ACTION Counter_Reset___entry:
NokCounter:=0;
(*Percent Register löschen*)
i:=0;
FOR i:=1 TO 100 BY 1 DO
  NokPercent[i]:= FALSE;
END_FOR
END_ACTION

ACTION Drehen_links_0_Grad__entry:
MP.ST02.TableData:=PushData(MP.ST02.TableData);
END_ACTION

ACTION Drehen_links_0_Grad__action:
ST02_62_Y6.MoveInit:=TRUE;
END_ACTION

ACTION Drehen_links_0_Grad__exit:
turn_done:=TRUE;
END_ACTION

ACTION Drehen_rechts_180_Grad___entry:
MP.ST02.TableData:=PushData(MP.ST02.TableData);
END_ACTION

ACTION Drehen_rechts_180_Grad___action:
ST02_62_Y6.MoveWork:=TRUE;
END_ACTION

ACTION Drehen_rechts_180_Grad___exit:
turn_done:=TRUE;
END_ACTION

ACTION Msg_Cam_Percent_entry:
MessageHandler.ClearMessageLines(sVisu:=Visu.Message);
END_ACTION

ACTION Msg_Cam_Percent_action:
MessageHandler.Msg.ID:='PM113';
MessageHandler.Msg.Name:='Sensopart Kam.-Erg. Prüfung  n.i.o:';
MessageHandler.Msg.Text:='Sensopart Kam.-Erg. Prüfung  n.i.o:% Fehler';
MessageHandler.Msg.Color:=Color.red;
MessageHandler.Msg.Station:=3;
MessageHandler.MsgButton1Text:='continue';

MessageHandler(
	Prio:=2, 								(*1=highest, .. , 4=lowest*)
	Btn1Addr:=ADR(MsgOk),				(*Address of Button1 , if Zero then Button is unvisible*)
	Btn2Addr:=0(*ADR(MsgCancel)*),			(*Address of Button2 , if Zero then Button is unvisible*)
	sVisu:=Visu.Message);
END_ACTION

ACTION Msg_Cam_Percent_exit:
MsgOk:=FALSE;
MsgCancel:=FALSE;
END_ACTION

ACTION JumpAutoStop__action:
IF ST02_AutoStop.State=STATE_WAIT
THEN
	ST02_AutoStop(Start:=TRUE);
END_IF
END_ACTION

ACTION JumpAutoStop__exit:
ST02_AutoStop.Start:=FALSE;
END_ACTION

ACTION SeqEnd_action:
SFCTime:=TIME_TO_DINT(TIME()-SFCTimeStart);
State:=STATE_WAIT;
END_ACTION

TRANSITION OK:
ST02_35_S31.BitInToCheck
END_TRANSITION

TRANSITION OK_:
NOT MP.ST02.DummyPruefung_93pol
END_TRANSITION

TRANSITION Kamera_betriebsbereit:
(NOT ST02_DT_95_A1.b_kamera_aktiv (*Kamera Farberkennung*)
OR
NOT ST02_DT_95_A1.sm_kamera_nicht_bb) 	 (*Kamera Farberkennung*)
AND
(NOT ST02_DT_95_A2.sm_kamera_nicht_bb
OR
NOT ST02_DT_95_A2.Activated)
END_TRANSITION

TRANSITION Drucker_bereit:
MP.ST02.DummyPruefung_93pol OR
ST00_72_X1_8.BitInToCheck 	(* Tampondrucker Bedruckung ausgeführt oder betriebsbereit *)
END_TRANSITION

TRANSITION MsgOk:
MsgOk OR

ST00_72_X1_8.BitInToCheck 	(* Tampondrucker Bedruckung ausgeführt oder betriebsbereit *)
END_TRANSITION

TRANSITION 180_Grad:
NOT ST02_DT_62_B81.ValveSensor AND	(* Tisch  0 Grad*)
ST02_DT_62_B91.ValveSensor				(* Tisch  180 Grad*)
END_TRANSITION

TRANSITION StateOk:
ST02_62_Y6.State=STATE_OK
AND
gTipImp
END_TRANSITION

TRANSITION nicht leer:
MP.ST02.TableData[2].ProcessData.Part AND

NOT ST02_DT_65B11.BitInToCheck					 (* Tampondrucker Nest 1 leer *)
END_TRANSITION

TRANSITION StateOk:
NOT ST02_Schwenkarm[1].b_180_grad AND
ST02_Schwenkarm[1].b_done
AND
gTipImp
END_TRANSITION

TRANSITION StateOk:
ST02_62_Y17.State=STATE_OK
AND
gTipImp
END_TRANSITION

TRANSITION Drucker_bereit:
NOT MP.ST02.DummyPruefung_93pol AND
ST00_72_X1_8.BitInToCheck 	(* Tampondrucker Bedruckung ausgeführt *)
END_TRANSITION

TRANSITION Drucker_busy:
NOT ST00_72_X1_8.BitInToCheck (* Tampondrucker Bedruckung ausgeführt *)
END_TRANSITION

TRANSITION not_busy:
ST00_72_X1_8.BitInToCheck (* Tampondrucker Bedruckung ausgeführt *)
END_TRANSITION

TRANSITION AutoStop:
		ModeSelect.Mode=MODE_AUTO_STOP
OR	ModeSelect.Mode=MODE_STEP_STOP
END_TRANSITION

TRANSITION Drucker_fertig:
ST00_72_X1_8.BitInToCheck (* Tampondrucker Bedruckung ausgeführt *)
END_TRANSITION

TRANSITION Dummypruefung:
MP.ST02.DummyPruefung_93pol
END_TRANSITION

TRANSITION aktiv:
ST02_DT_95_A1.b_kamera_aktiv (*Kamera Farberkennung*)
OR
ST02_DT_95_A2.Activated	(*Kamera Farberkennung Ethernet*)
END_TRANSITION

TRANSITION Busy:
ST02_DT_95_A1.b_busy	 (*Kamera Farberkennung*)
OR
ST02_DT_95_A2.st_ctrl_out.b_busy (*Kamera Farberkennung Ehternet*)
END_TRANSITION

TRANSITION Done:
(ST02_DT_95_A1.b_done AND	 (*Kamera Farberkennung*)
ST02_DT_95_A1.b_kamera_aktiv AND
((ST02_DT_95_A1.Ergebnis_IO AND NOT ST02_DT_95_A1.Ergebnis_NIO)OR
RepeatCounter>=2 ))
OR
(ST02_DT_95_A2.st_ctrl_out.b_fertig AND
ST02_DT_95_A2.Activated AND
((ST02_DT_95_A2.b_Kam_Pruef_IO AND NOT ST02_DT_95_A2.b_Kam_Pruef_NIO) OR
RepeatCounter>=2))
END_TRANSITION

TRANSITION CamNotAktiv:
(ST02_DT_95_A1.b_done	 (*Kamera Farberkennung*)
AND
NOT ST02_DT_95_A1.b_kamera_aktiv )
OR
(ST02_DT_95_A2.st_ctrl_out.b_fertig  (*Kamera Farberkennung Ethernet*)
AND
NOT ST02_DT_95_A2.Activated)
OR
(NOT ST02_DT_95_A1.b_kamera_aktiv AND NOT ST02_DT_95_A2.Activated)
END_TRANSITION

TRANSITION CamDone:
ST02_DT_95_A1.b_done	 (*Kamera Farberkennung*)
OR
ST02_DT_95_A2.st_ctrl_out.b_fertig	 (*Kamera Farberkennung Ethernet*)
END_TRANSITION

TRANSITION StateOk:
ST02_62_Y17.State=STATE_OK
AND
gTipImp
END_TRANSITION

TRANSITION StateOk:
NOT ST02_Schwenkarm[1].b_0_grad AND
ST02_Schwenkarm[1].b_done
AND
gTipImp
END_TRANSITION

TRANSITION Drucker_bereit:
NOT MP.ST02.DummyPruefung_93pol AND
ST00_72_X1_8.BitInToCheck (* Tampondrucker Bedruckung ausgeführt *)
END_TRANSITION

TRANSITION Drucker_busy:
NOT ST00_72_X1_8.BitInToCheck (* Tampondrucker Bedruckung ausgeführt *)
END_TRANSITION

TRANSITION not_busy:
ST00_72_X1_8.BitInToCheck (* Tampondrucker Bedruckung ausgeführt *)
END_TRANSITION

TRANSITION AutoStop:
		ModeSelect.Mode=MODE_AUTO_STOP
OR	ModeSelect.Mode=MODE_STEP_STOP
END_TRANSITION

TRANSITION Drucker_fertig:
ST00_72_X1_8.BitInToCheck (* Tampondrucker Bedruckung ausgeführt *)
END_TRANSITION

TRANSITION Dummypruefung:
MP.ST02.DummyPruefung_93pol
END_TRANSITION

TRANSITION aktiv:
ST02_DT_95_A1.b_kamera_aktiv (*Kamera Farberkennung*)
OR
ST02_DT_95_A2.Activated(*Kamera Farberkennung Ethernet*)
END_TRANSITION

TRANSITION Busy:
ST02_DT_95_A1.b_busy	 (*Kamera Farberkennung*)
OR
ST02_DT_95_A2.st_ctrl_out.b_busy	(*Kamera Farberkennung Ethernet*)
END_TRANSITION

TRANSITION Done:
ST02_DT_95_A1.b_done AND	 (*Kamera Farberkennung*)
ST02_DT_95_A1.b_kamera_aktiv AND
((ST02_DT_95_A1.Ergebnis_IO AND NOT ST02_DT_95_A1.Ergebnis_NIO)OR
RepeatCounter>=2 )
OR
(ST02_DT_95_A2.st_ctrl_out.b_fertig AND
ST02_DT_95_A2.Activated AND
((ST02_DT_95_A2.b_Kam_Pruef_IO AND NOT ST02_DT_95_A2.b_Kam_Pruef_NIO) OR
RepeatCounter>=2))
END_TRANSITION

TRANSITION CamNotAktiv:
(ST02_DT_95_A1.b_done	 (*Kamera Farberkennung*)
AND
NOT ST02_DT_95_A1.b_kamera_aktiv)
OR
(ST02_DT_95_A2.st_ctrl_out.b_fertig  (*Kamera Farberkennung Ethernet*)
AND
NOT ST02_DT_95_A2.Activated)
END_TRANSITION

TRANSITION CamDone:
ST02_DT_95_A1.b_done	 (*Kamera Farberkennung*)
OR
ST02_DT_95_A2.st_ctrl_out.b_fertig	 (*Kamera Farberkennung Ethernet*)
END_TRANSITION

TRANSITION StateOk:
NOT ST02_Schwenkarm[1].b_90_grad AND
ST02_Schwenkarm[1].b_done
AND
gTipImp
END_TRANSITION

TRANSITION 0_Grad:
ST02_DT_62_B81.ValveSensor AND	(* Tisch 0 Grad*)
NOT ST02_DT_62_B91.ValveSensor	(* Tisch 180 Grad*)
END_TRANSITION

TRANSITION StateOk:
ST02_62_Y6.State=STATE_OK
AND
gTipImp
END_TRANSITION

TRANSITION nicht leer:
MP.ST02.TableData[2].ProcessData.Part AND

NOT ST02_DT_65B21.BitInToCheck					 (* Tampondrucker Nest 2 leer *)
END_TRANSITION

TRANSITION StateOk:
NOT ST02_Schwenkarm[2].b_180_grad AND
ST02_Schwenkarm[2].b_done
AND
gTipImp
END_TRANSITION

TRANSITION StateOk:
ST02_62_Y18.State=STATE_OK
AND
gTipImp
END_TRANSITION

TRANSITION Drucker_bereit:
NOT MP.ST02.DummyPruefung_93pol AND
ST00_72_X1_8.BitInToCheck (* Tampondrucker Bedruckung ausgeführt *)
END_TRANSITION

TRANSITION Drucker_busy:
NOT ST00_72_X1_8.BitInToCheck (* Tampondrucker Bedruckung ausgeführt *)
END_TRANSITION

TRANSITION not_busy:
ST00_72_X1_8.BitInToCheck (* Tampondrucker Bedruckung ausgeführt *)
END_TRANSITION

TRANSITION AutoStop:
		ModeSelect.Mode=MODE_AUTO_STOP
OR	ModeSelect.Mode=MODE_STEP_STOP
END_TRANSITION

TRANSITION Drucker_fertig:
ST00_72_X1_8.BitInToCheck (* Tampondrucker Bedruckung ausgeführt *)
END_TRANSITION

TRANSITION Dummypruefung:
MP.ST02.DummyPruefung_93pol
END_TRANSITION

TRANSITION aktiv:
ST02_DT_95_A1.b_kamera_aktiv (*Kamera Farberkennung*)
OR
ST02_DT_95_A2.Activated	(*Kamera Farberkennung Ethernet*)
END_TRANSITION

TRANSITION Busy:
ST02_DT_95_A1.b_busy	 (*Kamera Farberkennung*)
OR
ST02_DT_95_A2.st_ctrl_out.b_busy (*Kamera Farberkennung Ehternet*)
END_TRANSITION

TRANSITION Done:
(ST02_DT_95_A1.b_done AND	 (*Kamera Farberkennung*)
ST02_DT_95_A1.b_kamera_aktiv AND
((ST02_DT_95_A1.Ergebnis_IO AND NOT ST02_DT_95_A1.Ergebnis_NIO)OR
RepeatCounter>=2))
OR
(ST02_DT_95_A2.st_ctrl_out.b_fertig AND
ST02_DT_95_A2.Activated AND
((ST02_DT_95_A2.b_Kam_Pruef_IO AND NOT ST02_DT_95_A2.b_Kam_Pruef_NIO) OR
RepeatCounter>=2))
END_TRANSITION

TRANSITION CamNotAktiv:
(ST02_DT_95_A1.b_done	 (*Kamera Farberkennung*)
AND
NOT ST02_DT_95_A1.b_kamera_aktiv)
OR
(ST02_DT_95_A2.st_ctrl_out.b_fertig  (*Kamera Farberkennung Ethernet*)
AND
NOT ST02_DT_95_A2.Activated)
END_TRANSITION

TRANSITION CamDone:
ST02_DT_95_A1.b_done	 (*Kamera Farberkennung*)
OR
ST02_DT_95_A2.st_ctrl_out.b_fertig	 (*Kamera Farberkennung Ethernet*)
END_TRANSITION

TRANSITION StateOk:
ST02_62_Y18.State=STATE_OK
AND
gTipImp
END_TRANSITION

TRANSITION StateOk:
NOT ST02_Schwenkarm[2].b_0_grad AND
ST02_Schwenkarm[2].b_done
AND
gTipImp
END_TRANSITION

TRANSITION Drucker_bereit:
NOT MP.ST02.DummyPruefung_93pol AND
ST00_72_X1_8.BitInToCheck (* Tampondrucker Bedruckung ausgeführt *)
END_TRANSITION

TRANSITION Drucker_busy:
NOT ST00_72_X1_8.BitInToCheck (* Tampondrucker Bedruckung ausgeführt *)
END_TRANSITION

TRANSITION not_busy:
ST00_72_X1_8.BitInToCheck (* Tampondrucker Bedruckung ausgeführt *)
END_TRANSITION

TRANSITION AutoStop:
		ModeSelect.Mode=MODE_AUTO_STOP
OR	ModeSelect.Mode=MODE_STEP_STOP
END_TRANSITION

TRANSITION Drucker_fertig:
ST00_72_X1_8.BitInToCheck (* Tampondrucker Bedruckung ausgeführt *)
END_TRANSITION

TRANSITION Dummypruefung:
MP.ST02.DummyPruefung_93pol
END_TRANSITION

TRANSITION aktiv:
ST02_DT_95_A1.b_kamera_aktiv (*Kamera Farberkennung*)
OR
ST02_DT_95_A2.Activated (*Kamera Farberkennung Ethernet*)
END_TRANSITION

TRANSITION Busy:
ST02_DT_95_A1.b_busy	 (*Kamera Farberkennung*)
OR
ST02_DT_95_A2.st_ctrl_out.b_busy	(*Kamera Farberkennung Ethernet*)
END_TRANSITION

TRANSITION Done:
(ST02_DT_95_A1.b_done AND	 (*Kamera Farberkennung*)
ST02_DT_95_A1.b_kamera_aktiv AND
((ST02_DT_95_A1.Ergebnis_IO AND NOT ST02_DT_95_A1.Ergebnis_NIO)OR
RepeatCounter>=2 ))
OR
(ST02_DT_95_A2.st_ctrl_out.b_fertig AND
ST02_DT_95_A2.Activated AND
((ST02_DT_95_A2.b_Kam_Pruef_IO AND NOT ST02_DT_95_A2.b_Kam_Pruef_NIO) OR
RepeatCounter>=2))
END_TRANSITION

TRANSITION CamNotAktiv:
(ST02_DT_95_A1.b_done	 (*Kamera Farberkennung*)
AND
NOT ST02_DT_95_A1.b_kamera_aktiv)
OR
(ST02_DT_95_A2.st_ctrl_out.b_fertig  (*Kamera Farberkennung Ethernet*)
AND
NOT ST02_DT_95_A2.Activated)
END_TRANSITION

TRANSITION CamDone:
ST02_DT_95_A1.b_done	 (*Kamera Farberkennung*)
OR
ST02_DT_95_A2.st_ctrl_out.b_fertig	 (*Kamera Farberkennung Ethernet*)
END_TRANSITION

TRANSITION StateOk:
NOT ST02_Schwenkarm[2].b_90_grad AND
ST02_Schwenkarm[2].b_done
AND
 (gTipImp OR ModeSelect.Mode=MODE_MANUAL)
END_TRANSITION

TRANSITION CounterOK:
NOT MP.ST02.DummyPruefung_93pol AND
NokCounter<MP.ST02.CamNoOfErrors AND
NokCounterPercent < MP.ST02.CamNoOfErrorsPercent
OR
( MP.ST02.DummyPruefung_93pol AND
LoopCounter < 6)
END_TRANSITION

TRANSITION Nok_Cont:
NOT MP.ST02.DummyPruefung_93pol AND
NokCounter >= MP.ST02.CamNoOfErrors
END_TRANSITION

TRANSITION Nok_Percent:
NOT MP.ST02.DummyPruefung_93pol AND
NokCounterPercent >= MP.ST02.CamNoOfErrorsPercent
END_TRANSITION

TRANSITION Dummytest:
 MP.ST02.DummyPruefung_93pol AND
LoopCounter = 6
END_TRANSITION

TRANSITION Robo_free:
Robot01.ActualArea <> 3
END_TRANSITION

TRANSITION 180_Grad_:
NOT ST02_DT_62_B81.ValveSensor AND	(* Tisch  0 Grad*)
ST02_DT_62_B91.ValveSensor				(* Tisch  180 Grad*)
END_TRANSITION

TRANSITION StateOk:
ST02_62_Y6.State=STATE_OK
AND
gTipImp
END_TRANSITION

TRANSITION 0_Grad_:
ST02_DT_62_B81.ValveSensor AND	(* Tisch 0 Grad*)
NOT ST02_DT_62_B91.ValveSensor	(* Tisch 180 Grad*)
END_TRANSITION

TRANSITION StateOk:
ST02_62_Y6.State=STATE_OK
AND
gTipImp
END_TRANSITION

TRANSITION end:
NOT MP.ST02.DummyPruefung_93pol
END_TRANSITION

TRANSITION AutoRun:
(ModeSelect.Mode=MODE_AUTO_RUN OR
ModeSelect.Mode=MODE_STEP_RUN)
OR (SpecialMode06.State=State_Run AND
		(gTypeCode=312 OR			(*93pol*)
		gTypeCode=499))				(*102pol*)
END_TRANSITION

TRANSITION AutoStop:
ModeSelect.Mode=MODE_AUTO_STOP OR
ModeSelect.Mode=MODE_STEP_STOP
END_TRANSITION

TRANSITION StateOk:
ST02_AutoStop.State=STATE_OK
END_TRANSITION
END_PROGRAM

(* POU Stations/ST_02_RT_Tampondrucker/ST02_SFCs/ST02_AutoStop, SFC *)
PROGRAM ST02_AutoStop

VAR_OUTPUT
	SFCCurrentPOU			: STRING:='ST02_AutoStop';
	SFCCurrentStep			: STRING:='';
	SFCTime					: DINT;
	State   				: StateObject	:= STATE_WAIT;
	Result  				: StateResult;
END_VAR
VAR_INPUT
	Start					: BOOL;
END_VAR
VAR
	MsgOK					: BOOL;
	MsgCancel				: BOOL;
	SFCRun					: BOOL;
	SFCTimeStart			: TIME;
	(* Userdefinded area *)

END_VAR
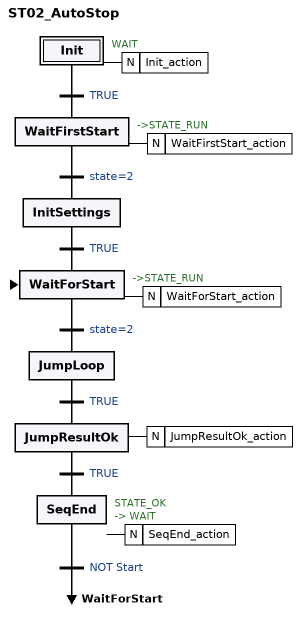
INITIAL_STEP Init: (* WAIT *)
	Init_action(N);
END_STEP
TRANSITION FROM Init TO WaitFirstStart := TRUE;
END_TRANSITION
STEP WaitFirstStart: (* ->STATE_RUN *)
	WaitFirstStart_action(N);
END_STEP
TRANSITION FROM WaitFirstStart TO InitSettings := state=2;
END_TRANSITION
STEP InitSettings:
END_STEP
TRANSITION FROM InitSettings TO WaitForStart := TRUE;
END_TRANSITION
STEP WaitForStart: (* ->STATE_RUN *)
	WaitForStart_action(N);
END_STEP
TRANSITION FROM WaitForStart TO JumpLoop := state=2;
END_TRANSITION
STEP JumpLoop:
END_STEP
TRANSITION FROM JumpLoop TO JumpResultOk := TRUE;
END_TRANSITION
STEP JumpResultOk:
	JumpResultOk_action(N);
END_STEP
TRANSITION FROM JumpResultOk TO SeqEnd := TRUE;
END_TRANSITION
STEP SeqEnd: (* STATE_OK / -> WAIT *)
	SeqEnd_action(N);
END_STEP
TRANSITION FROM SeqEnd TO WaitForStart := NOT Start;
END_TRANSITION

ACTION Init_action:
Start:=FALSE;
State:=STATE_WAIT;
MsgOK:=FALSE;
MsgCancel:=FALSE;
SFCRun:=FALSE;
END_ACTION

ACTION WaitFirstStart_action:
IF Start
THEN
	State:=STATE_RUN;
	Result:=RESULT_NON;
(*ELSE*)
END_IF
END_ACTION

ACTION WaitForStart_action:
IF Start
THEN
	State:=STATE_RUN;
	Result:=RESULT_NON;
	SFCTimeStart:=TIME();
END_IF
END_ACTION

ACTION JumpResultOk_action:
Result:=RESULT_OK;
END_ACTION

ACTION SeqEnd_action:
IF 	State=STATE_RUN THEN
	SFCTime:=TIME_TO_DINT(TIME()-SFCTimeStart);
	State:=STATE_OK;
END_IF

IF 	NOT Start THEN
	State:=STATE_WAIT;
END_IF
END_ACTION
END_PROGRAM

(* POU Stations/ST_03_Ruestsaetze/ST_03_SFCs/Zufuehrungen/ST03_102pol_Zufuehrung, SFC *)
 PROGRAM ST03_102pol_Zufuehrung
VAR_OUTPUT
	SFCCurrentPOU			: STRING:='ST03_102pol_Zufuehrung';
	SFCCurrentStep			: STRING:='';
	FB_CurrentStepHistorie	: FB_CurrentStepHistorie;
	SFCTime					: DINT;
	State   				: StateObject	:= STATE_WAIT;
END_VAR
VAR_INPUT
	Start				: BOOL;
	Result  			: DINT;
END_VAR
VAR
	MsgOK				: BOOL;
	MsgCancel			: BOOL;
	SFCRun				: BOOL;
	SFCTimeStart		: TIME;
	(* Userdefinded area *)
	i					: INT;
	PartReady			: BOOL;

	ResultBufferIFM		: ARRAY[1..10] OF BOOL;
	LoopCounter			: DINT;	(* Anzahl Dummy *)
	Dummy_test_Result	: BOOL;
	Delay				: TON;
END_VAR
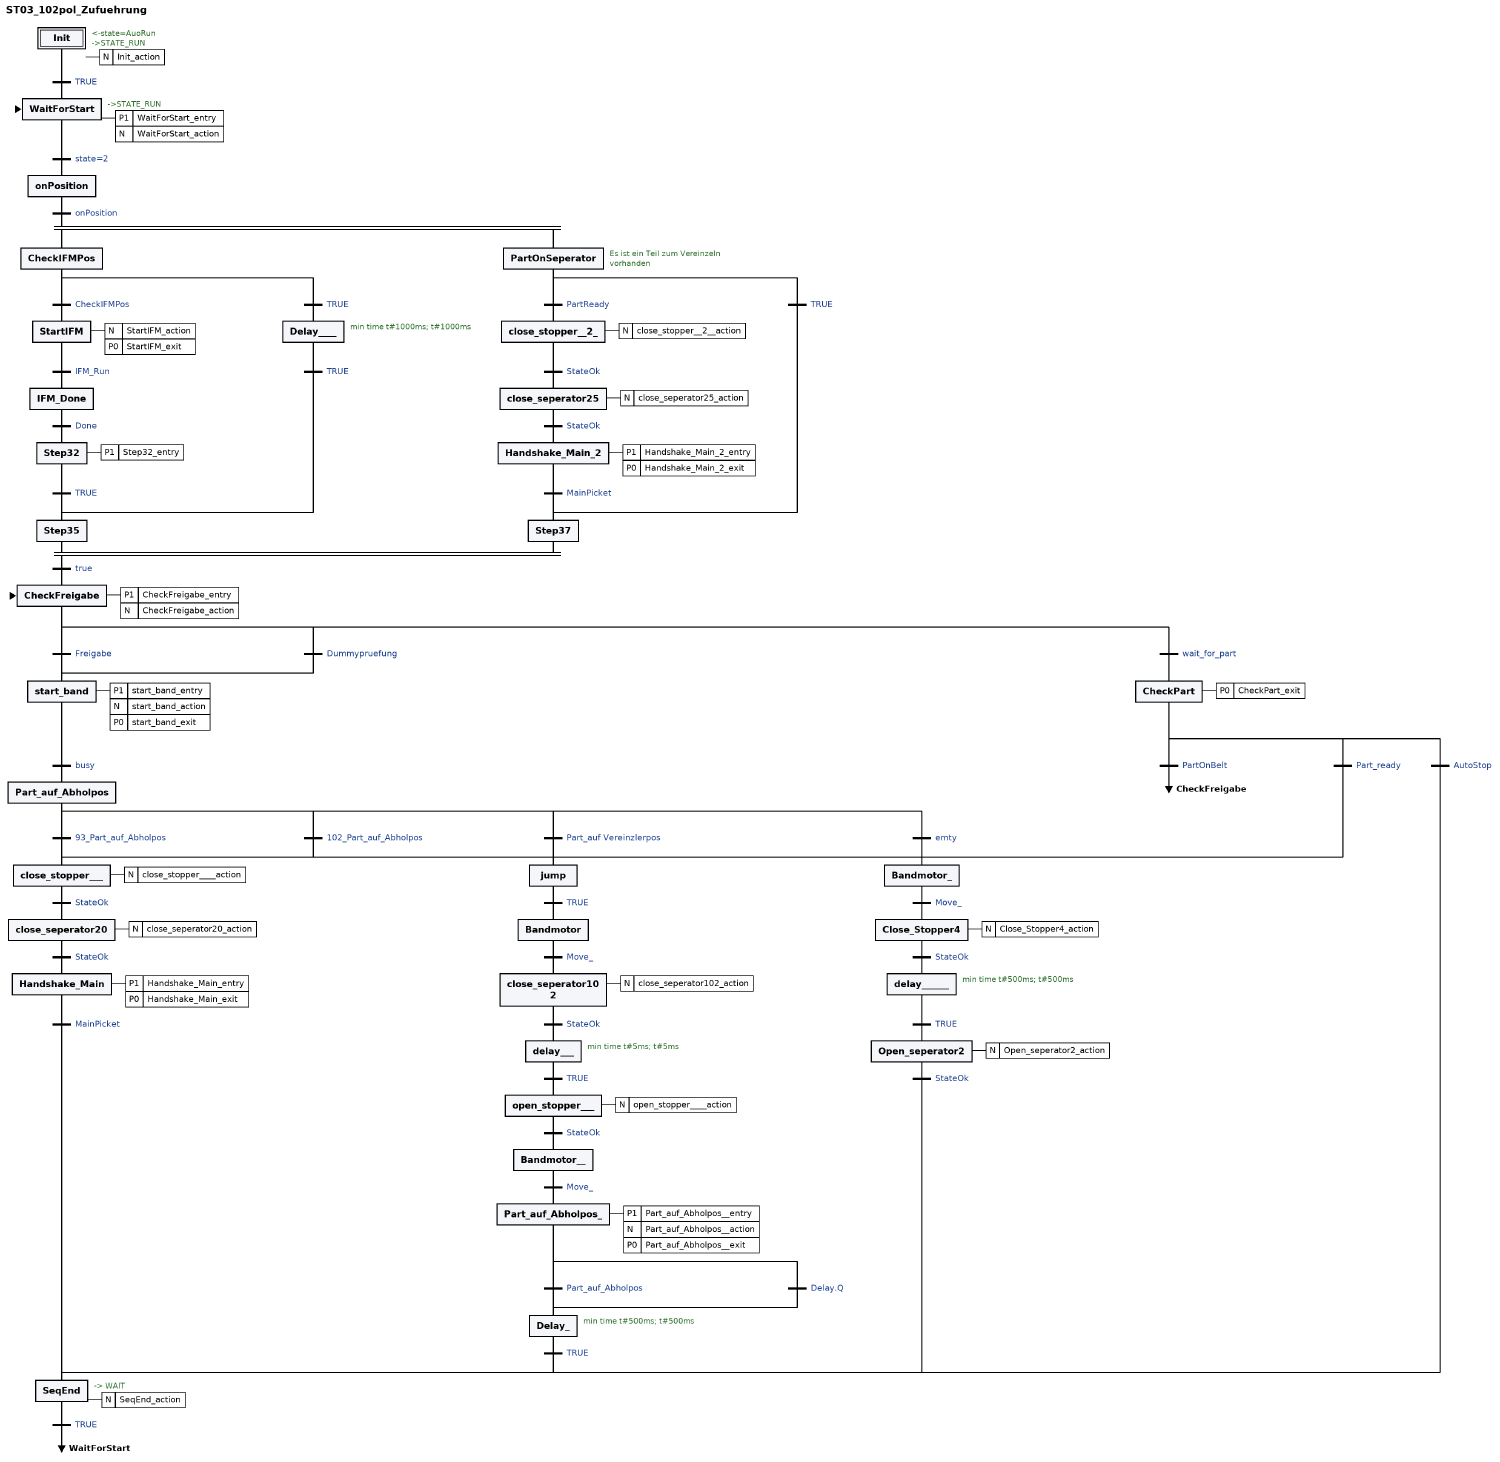
INITIAL_STEP Init: (* <-state=AuoRun / ->STATE_RUN *)
	Init_action(N);
END_STEP
TRANSITION FROM Init TO WaitForStart := TRUE;
END_TRANSITION
STEP WaitForStart: (* ->STATE_RUN *)
	WaitForStart_entry(P1);
	WaitForStart_action(N);
END_STEP
TRANSITION FROM WaitForStart TO onPosition := state=2;
END_TRANSITION
STEP onPosition:
END_STEP
TRANSITION FROM onPosition TO (CheckIFMPos, PartOnSeperator) := onPosition;
END_TRANSITION
STEP CheckIFMPos:
END_STEP
TRANSITION FROM CheckIFMPos TO StartIFM := CheckIFMPos;
END_TRANSITION
TRANSITION FROM CheckIFMPos TO Delay____ := TRUE;
END_TRANSITION
STEP Delay____: (* min time t#1000ms; t#1000ms *)
END_STEP
TRANSITION FROM Delay____ TO Step35 := TRUE;
END_TRANSITION
STEP StartIFM:
	StartIFM_action(N);
	StartIFM_exit(P0);
END_STEP
TRANSITION FROM StartIFM TO IFM_Done := IFM_Run;
END_TRANSITION
STEP IFM_Done:
END_STEP
TRANSITION FROM IFM_Done TO Step32 := Done;
END_TRANSITION
STEP Step32:
	Step32_entry(P1);
END_STEP
TRANSITION FROM Step32 TO Step35 := TRUE;
END_TRANSITION
STEP Step35:
END_STEP
STEP PartOnSeperator: (* Es ist ein Teil zum Vereinzeln vorhanden *)
END_STEP
TRANSITION FROM PartOnSeperator TO close_stopper__2_ := PartReady;
END_TRANSITION
TRANSITION FROM PartOnSeperator TO Step37 := TRUE;
END_TRANSITION
STEP close_stopper__2_:
	close_stopper__2__action(N);
END_STEP
TRANSITION FROM close_stopper__2_ TO close_seperator25 := StateOk;
END_TRANSITION
STEP close_seperator25:
	close_seperator25_action(N);
END_STEP
TRANSITION FROM close_seperator25 TO Handshake_Main_2 := StateOk;
END_TRANSITION
STEP Handshake_Main_2:
	Handshake_Main_2_entry(P1);
	Handshake_Main_2_exit(P0);
END_STEP
TRANSITION FROM Handshake_Main_2 TO Step37 := MainPicket;
END_TRANSITION
STEP Step37:
END_STEP
TRANSITION FROM (Step35, Step37) TO CheckFreigabe := true;
END_TRANSITION
STEP CheckFreigabe:
	CheckFreigabe_entry(P1);
	CheckFreigabe_action(N);
END_STEP
TRANSITION FROM CheckFreigabe TO start_band := Freigabe;
END_TRANSITION
TRANSITION FROM CheckFreigabe TO start_band := Dummypruefung;
END_TRANSITION
TRANSITION FROM CheckFreigabe TO CheckPart := wait_for_part;
END_TRANSITION
STEP CheckPart:
	CheckPart_exit(P0);
END_STEP
TRANSITION FROM CheckPart TO CheckFreigabe := PartOnBelt;
END_TRANSITION
TRANSITION FROM CheckPart TO close_stopper___ := Part_ready;
END_TRANSITION
TRANSITION FROM CheckPart TO SeqEnd := AutoStop;
END_TRANSITION
STEP start_band:
	start_band_entry(P1);
	start_band_action(N);
	start_band_exit(P0);
END_STEP
TRANSITION FROM start_band TO Part_auf_Abholpos := busy;
END_TRANSITION
STEP Part_auf_Abholpos:
END_STEP
TRANSITION FROM Part_auf_Abholpos TO close_stopper___ := 93_Part_auf_Abholpos;
END_TRANSITION
TRANSITION FROM Part_auf_Abholpos TO close_stopper___ := 102_Part_auf_Abholpos;
END_TRANSITION
TRANSITION FROM Part_auf_Abholpos TO jump := Part_auf Vereinzlerpos;
END_TRANSITION
TRANSITION FROM Part_auf_Abholpos TO Bandmotor_ := emty;
END_TRANSITION
STEP jump:
END_STEP
TRANSITION FROM jump TO Bandmotor := TRUE;
END_TRANSITION
STEP Bandmotor:
END_STEP
TRANSITION FROM Bandmotor TO close_seperator102 := Move_;
END_TRANSITION
STEP close_seperator102:
	close_seperator102_action(N);
END_STEP
TRANSITION FROM close_seperator102 TO delay___ := StateOk;
END_TRANSITION
STEP delay___: (* min time t#5ms; t#5ms *)
END_STEP
TRANSITION FROM delay___ TO open_stopper___ := TRUE;
END_TRANSITION
STEP open_stopper___:
	open_stopper____action(N);
END_STEP
TRANSITION FROM open_stopper___ TO Bandmotor__ := StateOk;
END_TRANSITION
STEP Bandmotor__:
END_STEP
TRANSITION FROM Bandmotor__ TO Part_auf_Abholpos_ := Move_;
END_TRANSITION
STEP Part_auf_Abholpos_:
	Part_auf_Abholpos__entry(P1);
	Part_auf_Abholpos__action(N);
	Part_auf_Abholpos__exit(P0);
END_STEP
TRANSITION FROM Part_auf_Abholpos_ TO Delay_ := Part_auf_Abholpos;
END_TRANSITION
TRANSITION FROM Part_auf_Abholpos_ TO Delay_ := Delay.Q;
END_TRANSITION
STEP Delay_: (* min time t#500ms; t#500ms *)
END_STEP
TRANSITION FROM Delay_ TO SeqEnd := TRUE;
END_TRANSITION
STEP Bandmotor_:
END_STEP
TRANSITION FROM Bandmotor_ TO Close_Stopper4 := Move_;
END_TRANSITION
STEP Close_Stopper4:
	Close_Stopper4_action(N);
END_STEP
TRANSITION FROM Close_Stopper4 TO delay______ := StateOk;
END_TRANSITION
STEP delay______: (* min time t#500ms; t#500ms *)
END_STEP
TRANSITION FROM delay______ TO Open_seperator2 := TRUE;
END_TRANSITION
STEP Open_seperator2:
	Open_seperator2_action(N);
END_STEP
TRANSITION FROM Open_seperator2 TO SeqEnd := StateOk;
END_TRANSITION
STEP close_stopper___:
	close_stopper____action(N);
END_STEP
TRANSITION FROM close_stopper___ TO close_seperator20 := StateOk;
END_TRANSITION
STEP close_seperator20:
	close_seperator20_action(N);
END_STEP
TRANSITION FROM close_seperator20 TO Handshake_Main := StateOk;
END_TRANSITION
STEP Handshake_Main:
	Handshake_Main_entry(P1);
	Handshake_Main_exit(P0);
END_STEP
TRANSITION FROM Handshake_Main TO SeqEnd := MainPicket;
END_TRANSITION
STEP SeqEnd: (* -> WAIT *)
	SeqEnd_action(N);
END_STEP
TRANSITION FROM SeqEnd TO WaitForStart := TRUE;
END_TRANSITION

ACTION Init_action:
Start:=FALSE;
State:=STATE_WAIT;
MsgOK:=FALSE;
MsgCancel:=FALSE;
SFCRun:=FALSE;
Result:=RESULT_NON;
PartReady := FALSE;
ST03_Band.fb_ton_Stopp_Band.IN:=FALSE;
LoopCounter :=0;
END_ACTION

ACTION WaitForStart_entry:
;
END_ACTION

ACTION WaitForStart_action:
IF 	Start   THEN
	State:=STATE_RUN;
	Result:=RESULT_NON;
	SFCTimeStart:=TIME();
	Start:=FALSE;
ELSE
	State:=STATE_WAIT;
	MsgOK:=FALSE;
	MsgCancel:=FALSE;
	SFCRun:=FALSE;
END_IF
END_ACTION

ACTION StartIFM_action:
ST03_IFM_Camera.Start:=TRUE;
END_ACTION

ACTION StartIFM_exit:
ST03_IFM_Camera.Start:=FALSE;
END_ACTION

ACTION Step32_entry:
IF ST02_FDB_55X1_6_IO.BitInToCheck AND
ST02_FDB_56X1_6_IO.BitInToCheck
THEN
   Dummy_test_Result:=TRUE;
ELSE
   Dummy_test_Result:=FALSE;
END_IF

(*Ergebnise in Puffer eintragen für Dummyprüfung IFM Kamera*)
i:=0;
FOR i:=10 TO 2 BY-1 DO
	ResultBufferIFM[i]:=ResultBufferIFM[i-1];
END_FOR
ResultBufferIFM[1]:=Dummy_test_Result;
END_ACTION

ACTION close_stopper__2__action:
ST00_74_Y2_4.MoveInit:=TRUE;
END_ACTION

ACTION close_seperator25_action:
ST00_74_Y2_5.MoveWork:=TRUE;
END_ACTION

ACTION Handshake_Main_2_entry:
PartReady := TRUE;
END_ACTION

ACTION Handshake_Main_2_exit:
PartReady := FALSE;
END_ACTION

ACTION CheckFreigabe_entry:
LoopCounter := LoopCounter +1;
END_ACTION

ACTION CheckFreigabe_action:
IF MP.ST02.DummyPruefung_93pol THEN
ST03_BG3_X53_0.SetSignalHigh := TRUE; (*LED Taster Start Band Dummyprüfung*)
END_IF
END_ACTION

ACTION CheckPart_exit:
ST03_Band.fb_ton_Stopp_Band.IN:=FALSE;
END_ACTION

ACTION start_band_entry:
IF NOT MP.ST02.DummyPruefung_93pol THEN
			ST03_51_M1.sVelo.maxRpm;
			ST03_51_M1.Vorgabe_Velo:=32000; 			(*mm/min*)
			ST03_51_M1.Vorgabe_Pos_Rel:=MP.ST02.IFMPos;
			ST03_51_M1.MoveRel:=TRUE;
ELSE
			ST03_51_M1.sVelo.maxRpm;
			ST03_51_M1.Vorgabe_Velo:=16000; 			(*mm/min*)
			ST03_51_M1.Vorgabe_Pos_Rel:=MP.ST02.IFMPosDummy;
			ST03_51_M1.MoveRel:=TRUE;
END_IF


ST03_Band.fb_ton_Stopp_Band.IN:=TRUE;
END_ACTION

ACTION start_band_action:
ST03_BG3_X53_0.SetSignalLow := TRUE; (*LED Taster Start Band Dummyprüfung*)
END_ACTION

ACTION start_band_exit:
ST03_51_M1.MoveRel:=FALSE;
END_ACTION

ACTION close_seperator102_action:
ST00_74_Y2_5.MoveWork:=TRUE;
END_ACTION

ACTION open_stopper____action:
ST00_74_Y2_4.MoveWork:=TRUE;
END_ACTION

ACTION Part_auf_Abholpos__entry:
Delay(IN:=FALSE);
END_ACTION

ACTION Part_auf_Abholpos__action:
Delay(IN:=TRUE, PT:=t#2s);
END_ACTION

ACTION Part_auf_Abholpos__exit:
Delay(IN:=FALSE);
END_ACTION

ACTION Close_Stopper4_action:
ST00_74_Y2_4.MoveInit:=TRUE;
END_ACTION

ACTION Open_seperator2_action:
ST00_74_Y2_5.MoveInit:=TRUE;
END_ACTION

ACTION close_stopper____action:
ST00_74_Y2_4.MoveInit:=TRUE;
END_ACTION

ACTION close_seperator20_action:
ST00_74_Y2_5.MoveWork:=TRUE;
END_ACTION

ACTION Handshake_Main_entry:
PartReady := TRUE;
END_ACTION

ACTION Handshake_Main_exit:
PartReady := FALSE;
END_ACTION

ACTION SeqEnd_action:
SFCTime:=TIME_TO_DINT(TIME()-SFCTimeStart);
State:=STATE_WAIT;
END_ACTION

TRANSITION onPosition:
ST03_51_M1.On_Position
END_TRANSITION

TRANSITION CheckIFMPos:
(MP.ST00.IFMCameraActive AND NOT MP.ST02.DummyPruefung_93pol)
OR
(MP.ST02.DummyPruefung_93pol AND
LoopCounter <= 6)
END_TRANSITION

TRANSITION IFM_Run:
ST03_IFM_Camera.State = STATE_RUN
END_TRANSITION

TRANSITION Done:
ST03_IFM_Camera.State = STATE_WAIT
END_TRANSITION

TRANSITION PartReady:
(gTypeCode=4991 AND				(*102pol*)
 ST02_FDB_80_B02.BitInToCheck)	(*Entnahmeposition 2*)
OR
(gTypeCode=312 AND				(*93pol*)
 ST00_72_X1_3.BitInToCheck) 	(*Schnittstelle Tampondrucker Teil in Abholposition; Band Entnahmeposition 1*)
END_TRANSITION

TRANSITION StateOk:
ST00_74_Y2_4.State=STATE_OK
END_TRANSITION

TRANSITION StateOk:
ST00_74_Y2_5.State=STATE_OK
END_TRANSITION

TRANSITION MainPicket:
ST03_Main.Nest_Empty
END_TRANSITION

TRANSITION Freigabe:
NOT MP.ST02.DummyPruefung_93pol AND
NOT ST02_S1_40K01.BitInToCheck AND			(* Freigabe Förderband von SPM*)
NOT ST00_73_K4.BitInToCheck AND
(*Robot01.ActualArea <> 4	AND*)								(*  ISK anwesend am Vereinzler*)
NOT ST03_Band.fb_ton_Stopp_Band.Q
END_TRANSITION

TRANSITION Dummypruefung:
(SpecialMode06.StartErlaubt93pol AND
MP.ST02.DummyPruefung_93pol AND
NOT ST03_Band.fb_ton_Stopp_Band.Q AND
ST03_BG3_S53_0.BitInToCheck) (*Taster Start Band Dummyprüfung*)
OR
(SpecialMode06.StartErlaubt93pol AND
MP.ST02.DummyPruefung_93pol AND
LoopCounter >= 7 AND
NOT ST03_Band.fb_ton_Stopp_Band.Q)
END_TRANSITION

TRANSITION wait_for_part:
NOT MP.ST02.DummyPruefung_93pol
END_TRANSITION

TRANSITION PartOnBelt:
NOT ST02_FDB_40_B61.BitInToCheck
END_TRANSITION

TRANSITION Part_ready:
(gTypeCode=312 AND				(*93pol*)
 ST00_72_X1_3.BitInToCheck) 	(*Schnittstelle Tampondrucker Teil in Abholposition, Band Entnahmeposition 1 *)
OR
(gTypeCode=4991 AND				(*102pol*)
 ST02_FDB_80_B02.BitInToCheck)	(*Entnahmeposition 2*)
END_TRANSITION

TRANSITION AutoStop:
ModeSelect.Mode=MODE_AUTO_STOP OR
ModeSelect.Mode=MODE_STEP_STOP
END_TRANSITION

TRANSITION busy:
ST03_51_M1.Busy
END_TRANSITION

TRANSITION 93_Part_auf_Abholpos:
gTypeCode=312 AND			(*93pol*)
ST00_72_X1_3.BitInToCheck	(*Schnittstelle Tampondrucker Teil in Abholposition, Band Entnahmeposition 1 *)
END_TRANSITION

TRANSITION 102_Part_auf_Abholpos:
gTypeCode=4991 AND				(*102pol*)
ST02_FDB_80_B02.BitInToCheck	(*Entnahmeposition 2*)
END_TRANSITION

TRANSITION Part_auf Vereinzlerpos:
ST00_72_X1_3.BitInToCheck (* Schnittstelle Tampondrucker Teil in Abholposition *) (* Band Entnahmeposition 1 *)
END_TRANSITION

TRANSITION Move_:
NOT ST03_51_M1.On_Position
END_TRANSITION

TRANSITION StateOk:
ST00_74_Y2_5.State=STATE_OK
END_TRANSITION

TRANSITION StateOk:
ST00_74_Y2_4.State=STATE_OK
END_TRANSITION

TRANSITION Move_:
NOT ST03_51_M1.On_Position
END_TRANSITION

TRANSITION Part_auf_Abholpos:
ST02_FDB_80_B02.BitInToCheck 		(*Entnahmeposition 2*)
END_TRANSITION

TRANSITION emty:
NOT ST00_72_X1_3.BitInToCheck (* Schnittstelle Tampondrucker Teil in Abholposition *) (* Band Entnahmeposition 1 *)
END_TRANSITION

TRANSITION Move_:
NOT ST03_51_M1.On_Position
END_TRANSITION

TRANSITION StateOk:
ST00_74_Y2_4.State=STATE_OK
END_TRANSITION

TRANSITION StateOk:
ST00_74_Y2_5.State=STATE_OK
END_TRANSITION

TRANSITION StateOk:
ST00_74_Y2_4.State=STATE_OK
END_TRANSITION

TRANSITION StateOk:
ST00_74_Y2_5.State=STATE_OK
END_TRANSITION

TRANSITION MainPicket:
ST03_Main.Nest_Empty
END_TRANSITION
END_PROGRAM

(* POU Stations/ST_03_Ruestsaetze/ST_03_SFCs/ST03_IFM_Camera, SFC *)
PROGRAM ST03_IFM_Camera
VAR_OUTPUT
	SFCCurrentPOU		: STRING:='ST03_IFM_Camera';
	SFCCurrentStep		: STRING:='';
	FB_CurrentStepHistorie: FB_CurrentStepHistorie;
	SFCTime				: DINT;
	State   			: StateObject	:= STATE_WAIT;
	Result  			: StateResult;
END_VAR
VAR_INPUT
	Start				: BOOL;
END_VAR
VAR
	MsgOK				: BOOL;
	MsgCancel			: BOOL;
	SFCRun				: BOOL;
	SFCTimeStart		: TIME;
	fb_r_trig_start		: R_TRIG;
	Error				: ErrorStruct;
	(* Userdefinded area *)
	PartReady      		: BOOL;
 	ErrorSep        	: BOOL;
	NokCounter    		: DINT;
	WdhCounter   		: DINT;
	oldPosition			: LREAL;
END_VAR
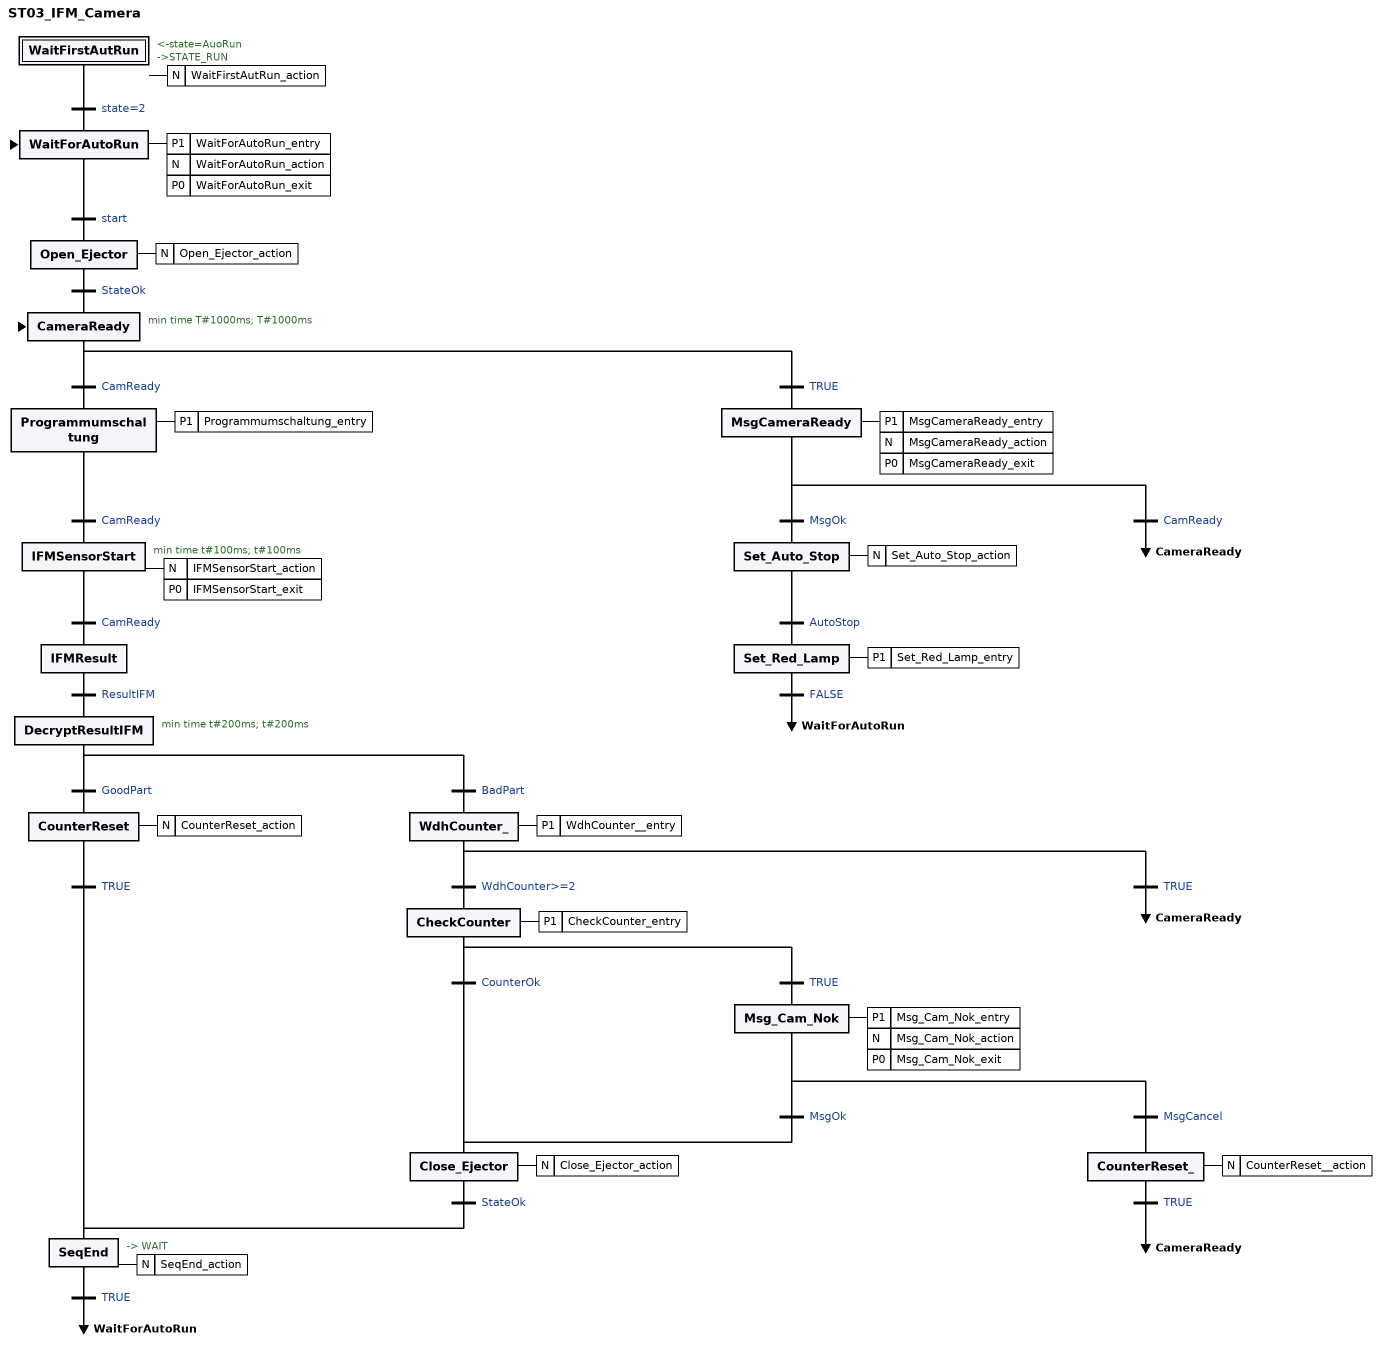
INITIAL_STEP WaitFirstAutRun: (* <-state=AuoRun / ->STATE_RUN *)
	WaitFirstAutRun_action(N);
END_STEP
TRANSITION FROM WaitFirstAutRun TO WaitForAutoRun := state=2;
END_TRANSITION
STEP WaitForAutoRun:
	WaitForAutoRun_entry(P1);
	WaitForAutoRun_action(N);
	WaitForAutoRun_exit(P0);
END_STEP
TRANSITION FROM WaitForAutoRun TO Open_Ejector := start;
END_TRANSITION
STEP Open_Ejector:
	Open_Ejector_action(N);
END_STEP
TRANSITION FROM Open_Ejector TO CameraReady := StateOk;
END_TRANSITION
STEP CameraReady: (* min time T#1000ms; T#1000ms *)
END_STEP
TRANSITION FROM CameraReady TO Programmumschaltung := CamReady;
END_TRANSITION
TRANSITION FROM CameraReady TO MsgCameraReady := TRUE;
END_TRANSITION
STEP MsgCameraReady:
	MsgCameraReady_entry(P1);
	MsgCameraReady_action(N);
	MsgCameraReady_exit(P0);
END_STEP
TRANSITION FROM MsgCameraReady TO Set_Auto_Stop := MsgOk;
END_TRANSITION
TRANSITION FROM MsgCameraReady TO CameraReady := CamReady;
END_TRANSITION
STEP Set_Auto_Stop:
	Set_Auto_Stop_action(N);
END_STEP
TRANSITION FROM Set_Auto_Stop TO Set_Red_Lamp := AutoStop;
END_TRANSITION
STEP Set_Red_Lamp:
	Set_Red_Lamp_entry(P1);
END_STEP
TRANSITION FROM Set_Red_Lamp TO WaitForAutoRun := FALSE;
END_TRANSITION
STEP Programmumschaltung:
	Programmumschaltung_entry(P1);
END_STEP
TRANSITION FROM Programmumschaltung TO IFMSensorStart := CamReady;
END_TRANSITION
STEP IFMSensorStart: (* min time t#100ms; t#100ms *)
	IFMSensorStart_action(N);
	IFMSensorStart_exit(P0);
END_STEP
TRANSITION FROM IFMSensorStart TO IFMResult := CamReady;
END_TRANSITION
STEP IFMResult:
END_STEP
TRANSITION FROM IFMResult TO DecryptResultIFM := ResultIFM;
END_TRANSITION
STEP DecryptResultIFM: (* min time t#200ms; t#200ms *)
END_STEP
TRANSITION FROM DecryptResultIFM TO CounterReset := GoodPart;
END_TRANSITION
TRANSITION FROM DecryptResultIFM TO WdhCounter_ := BadPart;
END_TRANSITION
STEP WdhCounter_:
	WdhCounter__entry(P1);
END_STEP
TRANSITION FROM WdhCounter_ TO CheckCounter := WdhCounter>=2;
END_TRANSITION
TRANSITION FROM WdhCounter_ TO CameraReady := TRUE;
END_TRANSITION
STEP CheckCounter:
	CheckCounter_entry(P1);
END_STEP
TRANSITION FROM CheckCounter TO Close_Ejector := CounterOk;
END_TRANSITION
TRANSITION FROM CheckCounter TO Msg_Cam_Nok := TRUE;
END_TRANSITION
STEP Msg_Cam_Nok:
	Msg_Cam_Nok_entry(P1);
	Msg_Cam_Nok_action(N);
	Msg_Cam_Nok_exit(P0);
END_STEP
TRANSITION FROM Msg_Cam_Nok TO Close_Ejector := MsgOk;
END_TRANSITION
TRANSITION FROM Msg_Cam_Nok TO CounterReset_ := MsgCancel;
END_TRANSITION
STEP CounterReset_:
	CounterReset__action(N);
END_STEP
TRANSITION FROM CounterReset_ TO CameraReady := TRUE;
END_TRANSITION
STEP Close_Ejector:
	Close_Ejector_action(N);
END_STEP
TRANSITION FROM Close_Ejector TO SeqEnd := StateOk;
END_TRANSITION
STEP CounterReset:
	CounterReset_action(N);
END_STEP
TRANSITION FROM CounterReset TO SeqEnd := TRUE;
END_TRANSITION
STEP SeqEnd: (* -> WAIT *)
	SeqEnd_action(N);
END_STEP
TRANSITION FROM SeqEnd TO WaitForAutoRun := TRUE;
END_TRANSITION

ACTION WaitFirstAutRun_action:
IF  ((ModeSelect.Mode=MODE_AUTO_RUN OR
	ModeSelect.Mode=MODE_STEP_RUN OR
	SpecialMode01.State=State_Run OR
	SpecialMode06.State=State_Run)
	AND
	(gTypeCode=312 OR	 (*93pol*)
	 gTypeCode=4991)	) (*102pol*)
THEN
	State:=STATE_RUN;
	Result:=RESULT_NON;
ELSE
	State:=STATE_WAIT;
END_IF

MsgOK:=FALSE;
MsgCancel:=FALSE;
SFCRun:=FALSE;
PartReady:=FALSE;
ErrorSep:=FALSE;

NokCounter:=0;
END_ACTION

ACTION WaitForAutoRun_entry:
State:=STATE_WAIT;
WdhCounter:=0;
END_ACTION

ACTION WaitForAutoRun_action:
fb_r_trig_start(CLK:=
		ST03_51_M1.On_Position AND	(*   Kamera ISK anwesend an Prüfposition  *)
		ABS(oldPosition - ST03_51_M1.sCtrl.in.Position) >10	 );
END_ACTION

ACTION WaitForAutoRun_exit:
State:=STATE_RUN;
Result:=RESULT_NON;
oldPosition:=ST03_51_M1.sCtrl.in.Position;
SFCTimeStart:=TIME();
END_ACTION

ACTION Open_Ejector_action:
ST02_62_Y4.MoveInit:=TRUE;
END_ACTION

ACTION MsgCameraReady_entry:
MessageHandler.ClearMessageLines(sVisu:=Visu.Message);
MsgOk := FALSE;
END_ACTION

ACTION MsgCameraReady_action:
IF	ST02_FDB_55X1_5_READY.BitInToCheck THEN				(*links*)
	MessageHandler.Msg.ID:='PM154';
ELSIF ST02_FDB_56X1_5_READY.BitInToCheck THEN 				(*rechts*)
	MessageHandler.Msg.ID:='PM155';
END_IF

MessageHandler.Msg.Name:='Kamera Ready';
MessageHandler.Msg.Text:= ' IFM Kamera nicht bereit ';
MessageHandler.Msg.Color:=Color.red;
MessageHandler.Msg.Station:=1;


MessageHandler(
	Prio:=2, 								(*1=highest, .. , 4=lowest*)
	Btn1Addr:=ADR(MsgOk),						(*Address of Button1 , if Zero then Button is unvisible*)
	Btn2Addr:=0,						(*Address of Button2 , if Zero then Button is unvisible*)
	sVisu:=Visu.Message);
END_ACTION

ACTION MsgCameraReady_exit:
MsgOk := FALSE;
END_ACTION

ACTION Set_Auto_Stop_action:
ModeSelect.AskForAutoStop:=TRUE;
END_ACTION

ACTION Set_Red_Lamp_entry:
ErrorSep:=TRUE;
END_ACTION

ACTION Programmumschaltung_entry:
ST02_FDB_55X1_7_JOB_BIT1.SetSignalHigh := TD.IFM_CamProgNo.0;	(* links *)
ST02_FDB_55X1_7_JOB_BIT1.SetSignalLow := NOT TD.IFM_CamProgNo.0;	(* links *)

ST02_FDB_55X1_7_JOB_BIT2.SetSignalHigh := TD.IFM_CamProgNo.1;	(* links *)
ST02_FDB_55X1_7_JOB_BIT2.SetSignalLow := NOT TD.IFM_CamProgNo.1;	(* links *)

ST02_FDB_56X1_7_JOB_BIT1.SetSignalHigh := TD.IFM_CamProgNo.0;	(* rechts *)
ST02_FDB_56X1_7_JOB_BIT1.SetSignalLow := NOT TD.IFM_CamProgNo.0;	(* rechts *)

ST02_FDB_56X1_7_JOB_BIT2.SetSignalHigh := TD.IFM_CamProgNo.1;	(* rechts *)
ST02_FDB_56X1_7_JOB_BIT2.SetSignalLow := NOT TD.IFM_CamProgNo.1;	(* rechts *)
END_ACTION

ACTION IFMSensorStart_action:
ST02_FDB_55X1_2_TRIGGER.SetSignalHigh := TRUE;
ST02_FDB_56X1_2_TRIGGER.SetSignalHigh := TRUE;
END_ACTION

ACTION IFMSensorStart_exit:
ST02_FDB_55X1_2_TRIGGER.SetSignalLow := TRUE;
ST02_FDB_56X1_2_TRIGGER.SetSignalLow := TRUE;
END_ACTION

ACTION WdhCounter__entry:
WdhCounter:=WdhCounter+1;
END_ACTION

ACTION CheckCounter_entry:
IF NOT MP.ST02.DummyPruefung_93pol AND
ST02_FDB_54_B41.BitInToCheck (*Schlechtteile werden nur hoch gezählt wenn der Sensor belegt ist*)
THEN
gNokPartsWingCam := gNokPartsWingCam+1;
NokCounter:=NokCounter+1;
END_IF
END_ACTION

ACTION Msg_Cam_Nok_entry:
MessageHandler.ClearMessageLines(sVisu:=Visu.Message);
END_ACTION

ACTION Msg_Cam_Nok_action:
MessageHandler.Msg.ID:='PM156';
MessageHandler.Msg.Name:='Fluegelerkennung:';
MessageHandler.Msg.Text:='Fluegelerkennung: Fehler in Folge Weiter mit "OK" Stop. mit "Abbrechen';
MessageHandler.Msg.Color:=Color.red;
MessageHandler.Msg.Station:=2;
MessageHandler.MsgButton1Text:='continue';

MessageHandler(
	Prio:=2, 						(*1=highest, .. , 4=lowest*)
	Btn1Addr:=ADR(MsgOk),		(*Address of Button1 , if Zero then Button is unvisible*)
	Btn2Addr:=ADR(MsgCancel),	(*Address of Button2 , if Zero then Button is unvisible*)
	sVisu:=Visu.Message);
END_ACTION

ACTION Msg_Cam_Nok_exit:
MsgOk:=FALSE;
MsgCancel:=FALSE;

NokCounter:=0;
END_ACTION

ACTION CounterReset__action:
NokCounter:=0;
END_ACTION

ACTION Close_Ejector_action:
ST02_62_Y4.MoveWork:=TRUE;
END_ACTION

ACTION CounterReset_action:
NokCounter:=0;
END_ACTION

ACTION SeqEnd_action:
SFCTime:=TIME_TO_DINT(TIME()-SFCTimeStart);
State:=STATE_WAIT;
END_ACTION

TRANSITION start:
(*fb_r_trig_start.Q*)
Start
END_TRANSITION

TRANSITION StateOk:
ST02_62_Y4.State=STATE_OK
END_TRANSITION

TRANSITION CamReady:
ST02_FDB_55X1_5_READY.BitInToCheck AND		(*links*)
ST02_FDB_56X1_5_READY.BitInToCheck			(*rechts*)
END_TRANSITION

TRANSITION CamReady:
ST02_FDB_55X1_5_READY.BitInToCheck AND		(*links*)
ST02_FDB_56X1_5_READY.BitInToCheck			(*rechts*)
END_TRANSITION

TRANSITION AutoStop:
		ModeSelect.Mode=MODE_AUTO_STOP
OR	ModeSelect.Mode=MODE_STEP_STOP
END_TRANSITION

TRANSITION CamReady:
ST02_FDB_55X1_5_READY.BitInToCheck AND
ST02_FDB_56X1_5_READY.BitInToCheck
END_TRANSITION

TRANSITION CamReady:
ST02_FDB_55X1_5_READY.BitInToCheck AND		(*links*)
ST02_FDB_56X1_5_READY.BitInToCheck			(*rechts*)
END_TRANSITION

TRANSITION ResultIFM:
(ST02_FDB_55X1_6_IO.BitInToCheck OR
ST02_FDB_55X1_6_NIO.BitInToCheck)
AND
(ST02_FDB_56X1_6_IO.BitInToCheck OR
 ST02_FDB_56X1_6_NIO.BitInToCheck)
END_TRANSITION

TRANSITION GoodPart:
(ST02_FDB_55X1_6_IO.BitInToCheck AND
ST02_FDB_56X1_6_IO.BitInToCheck)OR
MP.ST02.DummyPruefung_93pol
END_TRANSITION

TRANSITION BadPart:
TRUE
END_TRANSITION

TRANSITION WdhCounter>=2:
WdhCounter > 2
END_TRANSITION

TRANSITION CounterOk:
NokCounter <= MP.ST00.Cam_NoOfErrors
END_TRANSITION

TRANSITION StateOk:
ST02_62_Y4.State=STATE_OK
END_TRANSITION
END_PROGRAM

(* POU Stations/ST_03_Ruestsaetze/ST_03_PRGs/ST03_Band, ST *)
PROGRAM ST03_Band
VAR_INPUT
	b_MoveRel 		:BOOL;
	fb_ton_Stopp_Band					: TON;
	bLockBand : BOOL;
END_VAR
VAR
	b_PosBetrieb	:BOOL;
	fb_rTrig_Off		: R_TRIG;
	fb_rTrig_stop		: R_TRIG;
	fb_ton_Off			: TON;
	fb_ton_Off2			: TON;
	fb_rTrig_On			: R_TRIG;
	fb_ton_Stau			: TON;
	fb_rtrig_Stopp_Band	: R_TRIG;

	fb_rTrig_MoveRel	: R_TRIG;

	MsgOK				: BOOL;
	MsgCancel			: BOOL;
	lr_PT				: LREAL;
END_VAR
fb_ton_Stopp_Band(IN:= ,PT:=t#10m , Q=> , ET=> );																	(*Stop Wenn von der Sritzguss kein Teile kommen*)

fb_rtrig_Stopp_Band(CLK:=ST00_72_X1_3.BitInToCheck OR ST02_FDB_80_B02.BitInToCheck);
IF	fb_rtrig_Stopp_Band.Q THEN
	fb_ton_Stopp_Band.IN:=FALSE;
END_IF

(*Störung Oriental Motor bei SG-Maschine 3621*)
IF MP.ST03.SGM_3621 THEN
	IF NOT St03_V2.BitInToCheck THEN
		ST03_A5.SetSignalLow := TRUE;

		MessageHandler.Msg.ID:='PM101';
		MessageHandler.Msg.Color:=Color.red;
		MessageHandler.Msg.Name:='Error Förderband';
		MessageHandler.Msg.Text:='Störung Motor Oriental Förderband!';
		MessageHandler.Msg.Station:=3;

		MessageHandler(
			Prio:=2, 							(*1=highest, .. , 4=lowest*)
			Btn1Addr:=ADR(MsgOk),				(*Address of Button1 , if Zero then Button is unvisible*)
			Btn2Addr:=0(*ADR(MsgCancel)*),		(*Address of Button2 , if Zero then Button is unvisible*)
			sVisu:=Visu.Message);
	END_IF
END_IF
(*Motorregelung einschalten=========================================================== *)

IF NOT MP.ST03.SGM_3621 THEN
	IF  NOT ST03_51_M1.Error_ THEN
		IF	(NOT Safety_Fuses_AirPressure.SafetyOK OR gRunEmpty) AND
			ST03_51_M1.on THEN
			ST03_51_M1.MotorOff :=TRUE;
		END_IF

		IF	ModeSelect.Mode > MODE_MANUAL AND
			NOT gRunEmpty AND
			Safety_Fuses_AirPressure.SafetyOK AND
			NOT ST03_51_M1.on THEN
			ST03_51_M1.MotorOn :=TRUE;
		END_IF
	END_IF
END_IF

(*Fahren bis zu Flügelkamera Förderband============================================================ *)

IF	gTypeCode=312  OR		(*93pol*)
	gTypeCode=4991 THEN	(*102pol*)
	b_PosBetrieb:=TRUE;
	(*Impolsbetrieb Förderband============================================================ *)

	IF 	ST03_IFM_Camera.State=STATE_WAIT OR
 		ModeSelect.Mode>=MODE_MANUAL OR
		NOT MP.ST00.IFMCameraActive THEN

		fb_rTrig_MoveRel(CLK:= ST03_51_M1.Ready AND
								b_MoveRel);

		IF	fb_rTrig_MoveRel.Q THEN
			ST03_51_M1.sVelo.maxRpm;
			ST03_51_M1.Vorgabe_Velo:=16000; 			(*mm/min*)
			ST03_51_M1.Vorgabe_Pos_Rel:=MP.ST02.IFMPos;
			ST03_51_M1.MoveRel:=TRUE;
		END_IF

	END_IF

ELSE
	(*Dauerbetrieb Förderband============================================================ *)
	b_PosBetrieb:=FALSE;
	fb_ton_Off(IN:=	ST03_Init_Lockings.b_freiFuerSG, 	(*Stop Wenn von der SG-Maschine keine Teile kommen*)
					PT:=t#5m, Q=> , ET=> );

	IF  gTypeCode = 322 THEN (*160pol*)
		fb_ton_Off2(IN:=ST00_73_K3.BitOutToSet AND								(* Schnittstelle Förderband frei für Spritzmaschine*)
						ST03_422_B64_4.BitInToCheck AND						(* Teil auf Abholposition Roboter *)
						(Robot01.ActualArea<>4), PT:=t#5s , Q=> , ET=> ); 			(*anhalten wenn Roboter nicht in der WT Area ist, die Ablageposition leer und die Abholposition voll ist*)
	ELSE
		fb_ton_Off2(IN:=ST00_73_K3.BitOutToSet AND								(* Schnittstelle Förderband frei für Spritzmaschine*)
						ST08_412_B59_0.BitInToCheck AND						(* Teil auf Abholposition Roboter *)
						(Robot01.ActualArea<>4), PT:=t#3s , Q=> , ET=> ); 		(*anhalten wenn Roboter nicht in der WT Area ist, die Ablageposition leer und die Abholposition voll ist*)
	END_IF

	IF  MP.ST03.SGM_3621 THEN
		fb_ton_Stau.PT:=t#15s;
	ELSE
		lr_PT:=(112-MP.ST02.Override_Band) *0.25;
		fb_ton_Stau.PT:=LREAL_TO_TIME(lr_PT * 1000);
	END_IF

	fb_ton_Stau(IN:=	NOT ST03_Init_Lockings.b_freiFuerSG AND (* ST00_73_K3.BitOutToSet AND*)
						Robot01.ActualArea <> 4 AND
						(ModeSelect.Mode = MODE_AUTO_RUN OR ModeSelect.Mode = MODE_AUTO_STOP) ,
						Q=> , ET=>); 			(*Stop wenn Teile nach dem Ablegen nicht weiter gefördert werden*)


	fb_rTrig_Off(CLK:= ModeSelect.Mode<=MODE_MANUAL );

	fb_rTrig_stop(CLK:= ModeSelect.Mode<=MODE_MANUAL AND ST03_51_M1.sVisuAxis.BtnStop.Pressed );

	fb_rTrig_On(CLK:= 	ModeSelect.Mode>MODE_MANUAL AND
						Safety_Fuses_AirPressure.SafetyOK );

	IF NOT MP.ST03.SGM_3621 THEN
		IF	fb_rTrig_On.Q THEN
			ST03_51_M1.MotorOn:=TRUE;
		END_IF

		IF	ST03_51_M1.On THEN
			ST03_51_M1.MoveP:=MP.ST03.BandMoveP;
			ST03_51_M1.MoveN:=NOT MP.ST03.BandMoveP;
		END_IF

		IF 	NOT DummyTest_160pol AND
			(fb_rTrig_Off.Q OR
			fb_ton_Off2.Q OR
			fb_ton_Off.Q OR
			fb_ton_Stau.Q OR
			fb_rTrig_stop.Q OR
			bLockBand) THEN
			ST03_51_M1.MotorOn:=FALSE;
			ST03_51_M1.MotorOff:=TRUE;
			ST03_51_M1.MoveN:=FALSE;
			ST03_51_M1.MoveP:=FALSE;
		ELSIF
			DummyTest_160pol AND NOT SpecialMode06.startBand THEN
			ST03_51_M1.MotorOn:=FALSE;
			ST03_51_M1.MotorOff:=TRUE;
			ST03_51_M1.MoveN:=FALSE;
			ST03_51_M1.MoveP:=FALSE;
		END_IF
	ELSE

		(*Ansteuerung Oriental Motor bei SG-Maschine 3621*)

		IF	NOT Safety_Fuses_AirPressure.SafetyOK THEN
			ST03_A5.SetSignalLow:=TRUE;
			ST03_A5.SetSignalHigh :=FALSE;
		ELSIF
			fb_rTrig_Off.Q OR fb_ton_Off2.Q OR fb_ton_Stau.Q THEN
			ST03_A5.SetSignalLow := TRUE;
			ST03_A5.SetSignalHigh :=FALSE;
		ELSIF
			ModeSelect.Mode >MODE_MANUAL AND
			Safety_Fuses_AirPressure.SafetyOK THEN
			ST03_A5.SetSignalHigh :=TRUE;
			ST03_A5.SetSignalLow := FALSE;
		END_IF
	END_IF


END_IF
END_PROGRAM

(* POU Stations/ST_00/ST00_PRGs/Safety_Fuses_AirPressure, ST *)
PROGRAM Safety_Fuses_AirPressure

VAR_OUTPUT
	SafetyOK					: BOOL;
END_VAR

VAR
	i							: INT;
	fb_rTrig_DoorsClosed		: ARRAY[0..9] OF R_TRIG;
	fb_rTrig_EmergencyMessage	: ARRAY[0..4] OF R_TRIG;

	DoorOpen					: STRING;
  	EmergencyStop				: STRING;
	DoorMessage				: BOOL;
	EmergencyMessage			: BOOL;

	fb_rTrig_Message			: R_TRIG;
	sID							: STRING(10);
END_VAR
(* Ready for Control ON *)
gReadyForControlOn :=

						NOT ST00_220_S1.BitInToCheck AND
						NOT ST00_220_S2.BitInToCheck (*AND
						NOT ST00_229_S1.BitInToCheck AND	(*Einlauf*)
						NOT ST00_230_S1.BitInToCheck*) ;	(*Auslauf*)

SafetyOK:=
					gReadyForControlOn AND
					ST00_200_A1_A1.BitInToCheck; 		(* alle Not-Aus IO *)

(*Reset-Hardware-Button*)
gResetButton:=FALSE;

(*Quittierung Not-Aus*)

ST00_200_A1_E4.PulseTime:=500;

ST00_200_A1_E4.PulseOn :=
				Visu.ModeSelect.BtnReset.Pressed OR
				ST00_292_S3_RESET.BitInToCheck OR
				ST00_245_S3_RESET.BitInToCheck AND
				gReadyForControlOn
														;
(* Tür Meldungen Generieren *)
IF	NOT DoorMessage THEN
	IF  St00_220_S1.BitInToCheck THEN
		sID:='PM31';
		DoorOpen:='Schutztüre 1 geöffnet + 0-220_S1';
		DoorMessage:=TRUE;
	ELSIF
		St00_220_S2.BitInToCheck THEN
		sID:='PM32';
		DoorOpen:='Schutztüre 2 geöffnet + 0-220_S2';
		DoorMessage:=TRUE;
	ELSIF
		ST00_229_S1.BitInToCheck THEN
		sID:='PM35';
		DoorOpen:='Schutztüre 5 Einlauf geöffnet + 0-229_S1';
	   	DoorMessage:=TRUE;
	ELSIF
		ST00_230_S1.BitInToCheck THEN
		sID:='PM36';
		DoorOpen:='Schutztüre 6 Auslauf geöffnet + 0-230_S1';
		DoorMessage:=TRUE;
	ELSIF
		ST00_231_S1.BitInToCheck THEN
		sID:='PM37';
		DoorOpen:='Schutztüre 7 Panel geöffnet + 0-231_S1';
		DoorMessage:=TRUE;
	ELSIF
		ST00_232_S1.BitInToCheck THEN
		sID:='PM38';
		DoorOpen:='Schutztüre 8 Auslauf geöffnet + 0-232_S1';
		DoorMessage:=TRUE;
	ELSIF
		ST00_240_S1.BitInToCheck THEN
		sID:='PM39';
		DoorOpen:='Schutztüre 9 Spritzguss geöffnet + 0-240_S1';
		DoorMessage:=TRUE;
	END_IF
END_IF
(*Tür Meldungen zurücksetzen*)
fb_rTrig_DoorsClosed[0](CLK:=NOT ST00_232_S1.BitInToCheck);
fb_rTrig_DoorsClosed[1](CLK:=NOT ST00_231_S1.BitInToCheck);
fb_rTrig_DoorsClosed[2](CLK:=NOT ST00_230_S1.BitInToCheck);
fb_rTrig_DoorsClosed[3](CLK:=NOT ST00_229_S1.BitInToCheck);
fb_rTrig_DoorsClosed[4](CLK:=NOT ST00_220_S1.BitInToCheck);
fb_rTrig_DoorsClosed[5](CLK:=NOT ST00_220_S2.BitInToCheck);
fb_rTrig_DoorsClosed[6](CLK:=NOT ST00_240_S1.BitInToCheck AND NOT ST00_245_V3_RESET.SignalOut );
fb_rTrig_DoorsClosed[7](CLK:=FALSE);
fb_rTrig_DoorsClosed[8](CLK:=FALSE);
fb_rTrig_DoorsClosed[9](CLK:=FALSE);
FOR i:=0 TO 9 BY 1 DO
	IF	fb_rTrig_DoorsClosed[i].Q THEN
		DoorMessage:=FALSE;
	END_IF
END_FOR

(*Tür Meldungen anzeigen*)
fb_rTrig_Message(CLK:=DoorMessage OR EmergencyMessage );
IF	fb_rTrig_Message.Q THEN
	MessageHandler.ClearMessageLines(sVisu:=Visu.Message);
END_IF

IF  DoorMessage THEN
	MessageHandler.Msg.ID:=sID;
	MessageHandler.Msg.Name:='Saftey_Doors_Open';
	MessageHandler.Msg.Text:=DoorOpen;
	MessageHandler.Msg.Color:=Color.orange;
	MessageHandler.Msg.Station:=0;

	MessageHandler(
		Prio:=3, 			(*1=highest, .. , 4=lowest*)
		Btn1Addr:=0,	(*Address of Button1 , if Zero then Button is unvisible*)
		Btn2Addr:=0,	(*Address of Button2 , if Zero then Button is unvisible*)
		sVisu:=Visu.Message);
END_IF


(* Notaus Meldungen Generieren =======================================================*)
IF	NOT EmergencyMessage THEN
	IF 	ST03_210_S1.BitInToCheck THEN
		sID:='PM41';
		EmergencyStop:='ST00_210_S2 Not-Halt 1 Anlage ausgelöst';
		EmergencyMessage:=TRUE;
	ELSIF
		ST00_X4_16.BitInToCheck THEN
		sID:='PM42';
		EmergencyStop:='ST00_X4_16 Not-Halt 2 Anlage ausgelöst';
		EmergencyMessage:=TRUE;
	(*ELSIF
		ST08_210_S2.BitInToCheck THEN
		sID:='PM42';
		EmergencyStop:='ST08_210_S2 Not-Halt 2 Anlage ausgelöst';
	    EmergencyMessage:=TRUE;*)
	END_IF
END_IF
(* Notaus Meldungen zurücksetzen*)
fb_rTrig_EmergencyMessage[0](CLK:=NOT ST03_210_S1.BitInToCheck);
fb_rTrig_EmergencyMessage[1](CLK:=NOT ST00_X4_16.BitInToCheck);
fb_rTrig_EmergencyMessage[2](CLK:=NOT ST08_210_S2.BitInToCheck);
fb_rTrig_EmergencyMessage[3](CLK:=FALSE);
fb_rTrig_EmergencyMessage[4](CLK:=FALSE);
FOR i:=0 TO 4 BY 1 DO
	IF	fb_rTrig_EmergencyMessage[i].Q THEN
		EmergencyMessage:=FALSE;
	END_IF
END_FOR

(* Notaus Meldungen anzeigen*)
IF  EmergencyMessage THEN
	MessageHandler.Msg.ID:=sID;
	MessageHandler.Msg.Name:='Notaus gedrückt';
	MessageHandler.Msg.Text:=EmergencyStop;
	MessageHandler.Msg.Color:=Color.red;
	MessageHandler.Msg.Station:=0;

	MessageHandler(
		Prio:=2, 			(*1=highest, .. , 4=lowest*)
		Btn1Addr:=0,	(*Address of Button1 , if Zero then Button is unvisible*)
		Btn2Addr:=0,	(*Address of Button2 , if Zero then Button is unvisible*)
		sVisu:=Visu.Message);
END_IF
END_PROGRAM

(* POU Stations/ST_03_Ruestsaetze/ST_03_PRGs/ST03_Init_Lockings, ST *)
PROGRAM ST03_Init_Lockings
VAR
	PosOffsetValid		: BOOL;
	b_freiFuerSG		: BOOL;
END_VAR

VAR_OUTPUT
	InputExp_Robot01	: BOOL;
END_VAR
PosOffsetValid:=gTypeDataValid;
IF 	NOT gBasicManualMode THEN
	InputExp_Robot01:=TRUE;
ELSE
(* 	Robot01 Entladen ST03
	Lockings for Robot01 of FB_Epson*)
	InputExp_Robot01:=PosOffsetValid;
END_IF

(* Freigabe an die Spritzgußmaschine für das Ablegen auf das Förderband *)

IF	b_freiFuerSG THEN
	ST00_73_K3.SetSignalHigh := TRUE;
ELSE
	ST00_73_K3.SetSignalLow := TRUE;
END_IF

CASE  gTypeCode OF

360,489:	(*P360 74pol*)(*P379 91pol*)(*P489 168pol*)
	IF	 MP.ST03.SGM_3621 THEN
		b_freiFuerSG:=
		 	NOT ST03_421_B63_4.BitInToCheck AND
			NOT ST03_421_B63_5.BitInToCheck AND
			NOT ST03_421_B63_6.BitInToCheck;
	ELSE
		b_freiFuerSG:=
		 	NOT ST08_412_B58_4.BitInToCheck AND
			NOT ST08_412_B58_5.BitInToCheck AND
			NOT ST08_412_B58_6.BitInToCheck;
	END_IF

379:
	b_freiFuerSG:=
		 	NOT ST08_412_B58_4.BitInToCheck AND
			NOT ST08_412_B58_5.BitInToCheck;
			(*NOT ST08_412_B58_6.BitInToCheck;*)

4992:	(*P4992 35pol*)
	b_freiFuerSG:=
		NOT ST08_412_B58_4.BitInToCheck;

4991,312:		(*P312 93pol*)(*P4991 102pol*)
	b_freiFuerSG:=
		ST03_51_M1.On_Position AND
		ST02_FDB_40_B61.BitInToCheck AND
		ST02_FDB_40_B71.BitInToCheck;

4871:		(*P4871 154pol*)
	b_freiFuerSG:=
		NOT ST03_425_B67_4.BitInToCheck AND
		NOT ST03_425_B67_5.BitInToCheck AND
		NOT ST03_425_B67_6.BitInToCheck;

4872:		(*P4872 154 Rasterplatte*)
	b_freiFuerSG:=
		NOT ST03_418_B60_6.BitInToCheck AND
		NOT ST03_418_B60_7.BitInToCheck;

322:		(*P322 160 polig*)
	b_freiFuerSG:=
		NOT ST03_421_B63_4.BitInToCheck AND
		NOT ST03_421_B63_5.BitInToCheck AND
		NOT ST03_421_B63_6.BitInToCheck;

522:		(*P522.01S 206 polig*)
	b_freiFuerSG:=
		NOT ST03_435_B67_4.BitInToCheck;

550:		(*P550 92 polig*)
	b_freiFuerSG:=
		ST03_444_B69_4.BitInToCheck;

564:		(*P564 124 polig*)
	b_freiFuerSG:=
		ST03_451_B69_4.BitInToCheck;

569:		(*P569 46 polig*)
	b_freiFuerSG:=
		ST03_461_B69_4.BitInToCheck;

5632,5633:	(*P5631 NOX 5/6 polig*)
	b_freiFuerSG:=
		NOT ST03_4x2_B69_0.BitInToCheck;

5631:		(*P5631 NOX 4 polig*)
	b_freiFuerSG:=
		ST03_491_B69_0.BitInToCheck;

5731:		(*P573 88polig*)
	b_freiFuerSG:=
		ST03_501_B69_0.BitInToCheck;

5732:		(*P573 88polig AMG*)
	b_freiFuerSG:=
		ST03_521_B69_0.BitInToCheck;

575,5753,5754,5755:		(*P575 7polig*)
	b_freiFuerSG:=
		NOT ST03_512_XG1.BitInToCheck AND		(*Klemmer frei*)
		ST03_512_B69_2.ValveSensor AND		(* ISK Klemmer 1 auf° GST*)
		ST03_512_B69_4.ValveSensor AND		(* ISK Klemmer 2 auf° GST*)
		ST03_512_B69_6.ValveSensor;

5771:		(*P5771 120polig*)
	b_freiFuerSG:=
		ST03_531_B69_0.BitInToCheck;


5772:		(*P5772 21polig*)
	b_freiFuerSG:=
		ST03_536_B69_0.BitInToCheck;

580:		(*P580 191polig*)
	b_freiFuerSG:=
		ST03_541_B69_0.BitInToCheck;

5831:		(*P5831 72polig*)
	b_freiFuerSG:=
		ST03_546_B69_0.BitInToCheck;

5832:		(*P5832 48polig*)
	b_freiFuerSG:=
		ST03_551_B69_0.BitInToCheck;

5841, 4993:		(*P5841 268pol, 102pol neu*)
	b_freiFuerSG:=
		ST03_556_B69_0.BitInToCheck AND
	(	NOT ST03_556_B69_5.BitInToCheck OR	(* Führungsschiene Überwachung Staustrecke*)
		NOT ST03_556_B69_6. BitInToCheck) ;		(* ISK anwesend am Stopper*)

5842:		(*P5841 268poligRP*)
	b_freiFuerSG:=
		NOT ST03_565_B72_0.BitInToCheck AND		(*Klemmer 1 frei*)
		NOT ST03_565_B72_1.BitInToCheck AND		(*Klemmer 2 frei*)
		ST03_565_B72_2.ValveSensor AND			(* ISK Klemmer 1 offen° GST*)
		ST03_565_B72_4.ValveSensor AND			(* ISK Klemmer 2 offen° GST*)
		ST03_565_B72_7.ValveSensor;				(* ISK Klemmer schwenkern 180° GST*)

598:		(*P98 33polig*)
	b_freiFuerSG:=
		NOT ST03_571_B69_0.BitInToCheck AND
		NOT ST03_571_B69_1.BitInToCheck;


END_CASE
END_PROGRAM

(* POU Stations/ST_03_Ruestsaetze/ST_03_SFCs/Zufuehrungen/ST03_160pol_Zufuehrung, SFC *)
 PROGRAM ST03_160pol_Zufuehrung
VAR_OUTPUT
	SFCCurrentPOU			: STRING:='ST03_160pol_Zufuehrung';
	SFCCurrentStep			: STRING:='';
	FB_CurrentStepHistorie	: FB_CurrentStepHistorie;
	SFCTime					: DINT;
	State   				: StateObject	:= STATE_WAIT;
END_VAR
VAR_INPUT
	Start				: BOOL;
	Result160pol		: DINT;
	CamResult  			: DINT;
	CamResult2			: DINT;
	CamResult3			: DINT;
	b_Printer_Off		: BOOL;
END_VAR
VAR
	MsgOK				: BOOL;
	MsgCancel			: BOOL;
	SFCRun				: BOOL;
	SFCTimeStart		: TIME;
	(* Userdefinded area *)
	i					:INT;
	RepeatCounter		:INT;
	NokCounter			:INT;
	NokCounterPercent	:INT;
  	NokPercent   		:ARRAY[1..100] OF BOOL;
	PartOk				:BOOL;	(* Ergebnisvariable für aktuelles *)

END_VAR
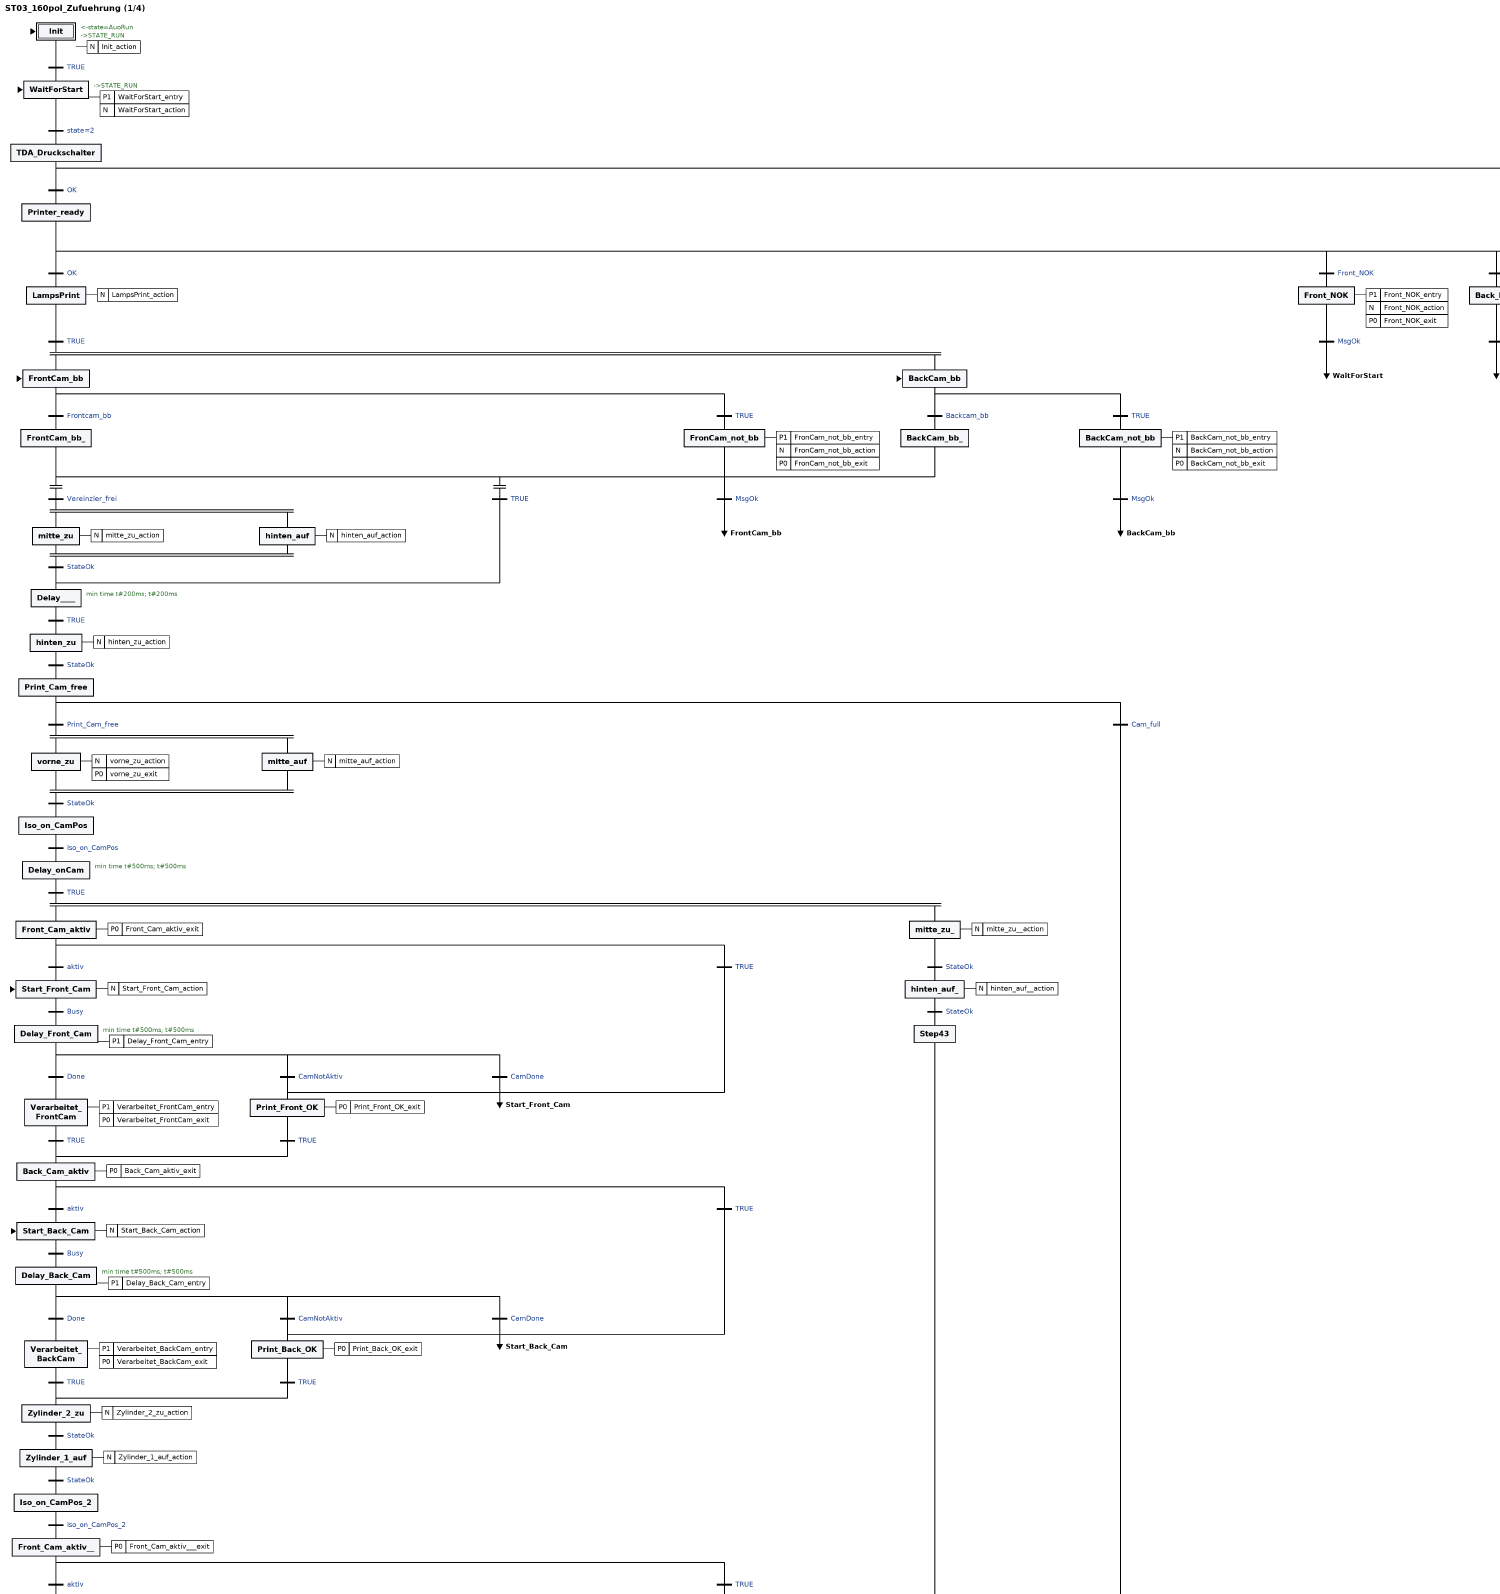
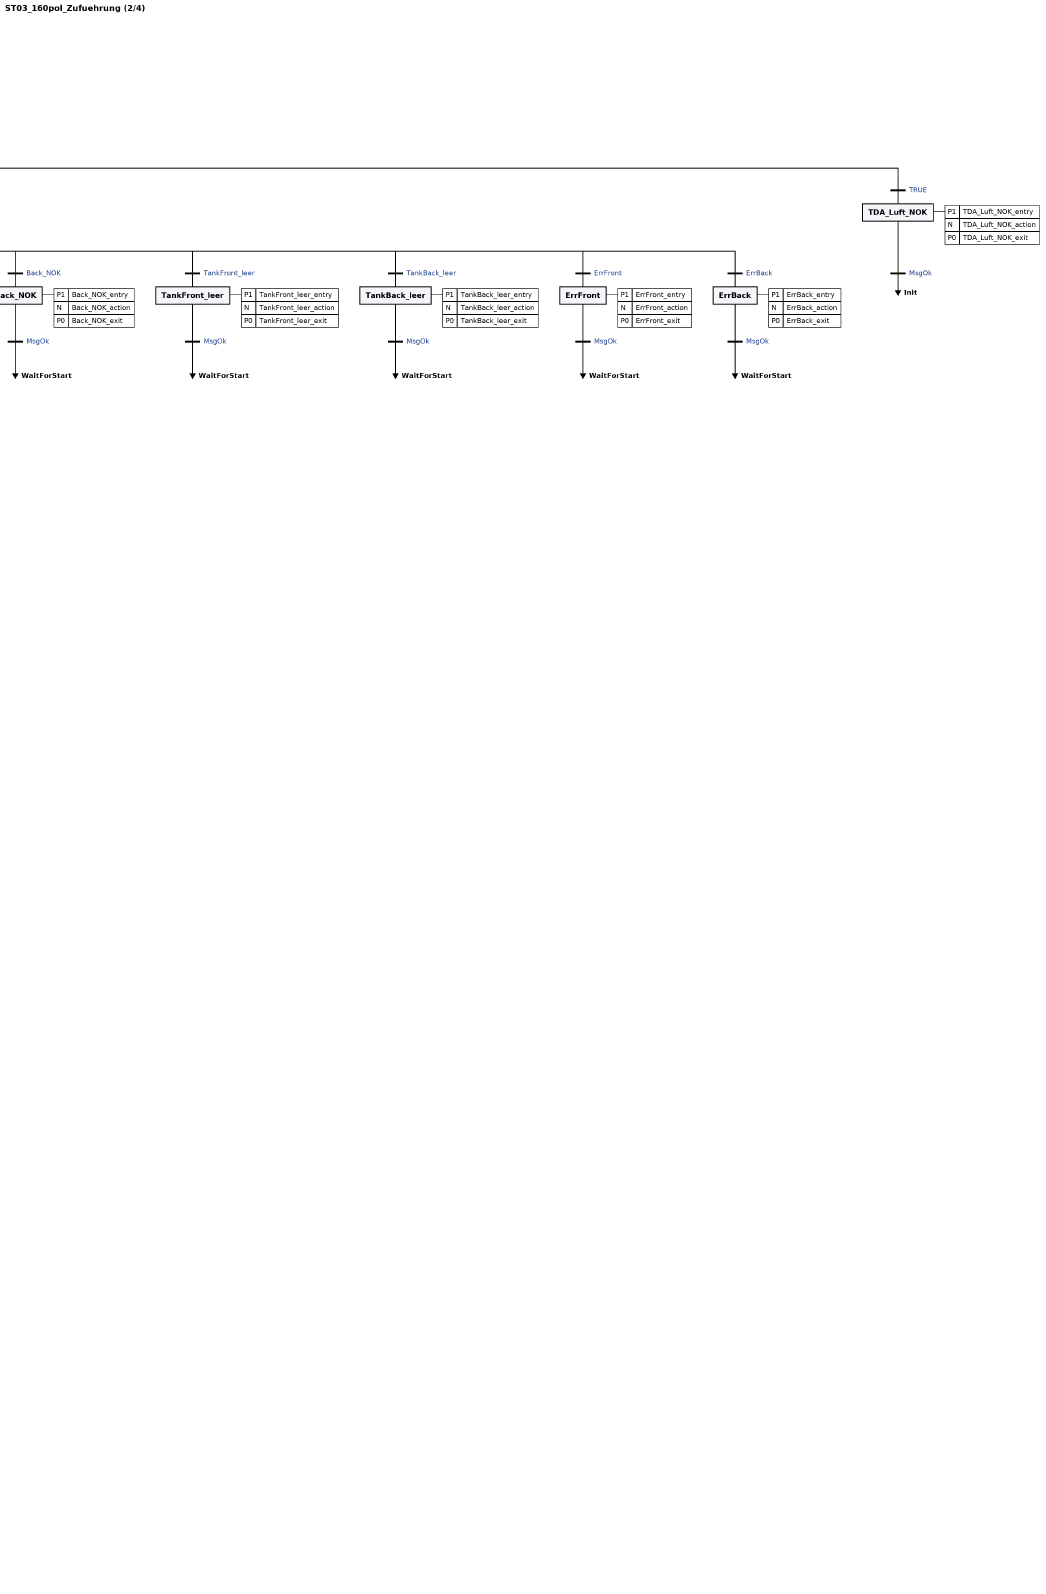
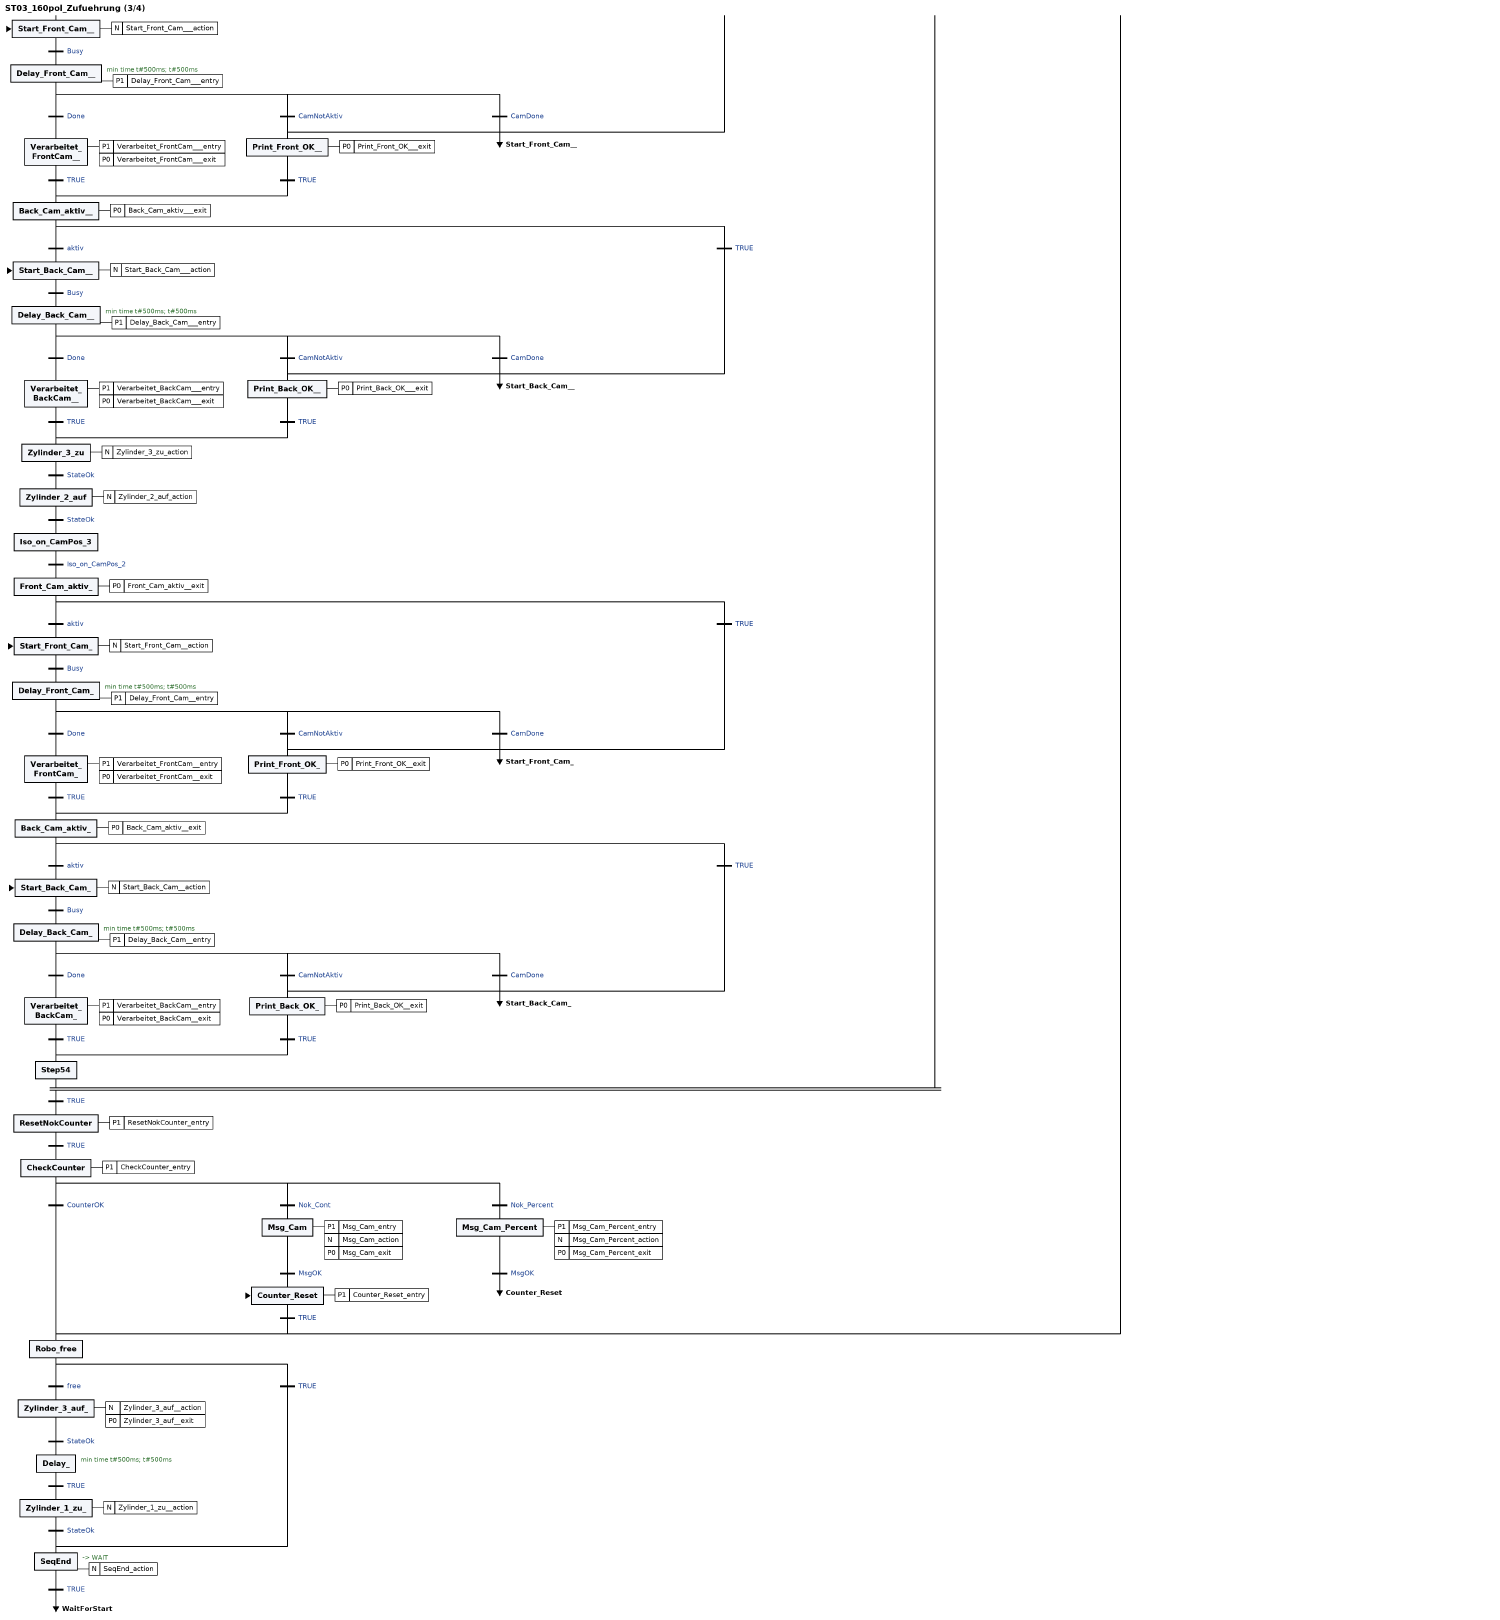
INITIAL_STEP Init: (* <-state=AuoRun / ->STATE_RUN *)
	Init_action(N);
END_STEP
TRANSITION FROM Init TO WaitForStart := TRUE;
END_TRANSITION
STEP WaitForStart: (* ->STATE_RUN *)
	WaitForStart_entry(P1);
	WaitForStart_action(N);
END_STEP
TRANSITION FROM WaitForStart TO TDA_Druckschalter := state=2;
END_TRANSITION
STEP TDA_Druckschalter:
END_STEP
TRANSITION FROM TDA_Druckschalter TO Printer_ready := OK;
END_TRANSITION
TRANSITION FROM TDA_Druckschalter TO TDA_Luft_NOK := TRUE;
END_TRANSITION
STEP TDA_Luft_NOK:
	TDA_Luft_NOK_entry(P1);
	TDA_Luft_NOK_action(N);
	TDA_Luft_NOK_exit(P0);
END_STEP
TRANSITION FROM TDA_Luft_NOK TO Init := MsgOk;
END_TRANSITION
STEP Printer_ready:
END_STEP
TRANSITION FROM Printer_ready TO LampsPrint := OK;
END_TRANSITION
TRANSITION FROM Printer_ready TO Front_NOK := Front_NOK;
END_TRANSITION
TRANSITION FROM Printer_ready TO Back_NOK := Back_NOK;
END_TRANSITION
TRANSITION FROM Printer_ready TO TankFront_leer := TankFront_leer;
END_TRANSITION
TRANSITION FROM Printer_ready TO TankBack_leer := TankBack_leer;
END_TRANSITION
TRANSITION FROM Printer_ready TO ErrFront := ErrFront;
END_TRANSITION
TRANSITION FROM Printer_ready TO ErrBack := ErrBack;
END_TRANSITION
STEP LampsPrint:
	LampsPrint_action(N);
END_STEP
TRANSITION FROM LampsPrint TO (FrontCam_bb, BackCam_bb) := TRUE;
END_TRANSITION
STEP Front_NOK:
	Front_NOK_entry(P1);
	Front_NOK_action(N);
	Front_NOK_exit(P0);
END_STEP
TRANSITION FROM Front_NOK TO WaitForStart := MsgOk;
END_TRANSITION
STEP Back_NOK:
	Back_NOK_entry(P1);
	Back_NOK_action(N);
	Back_NOK_exit(P0);
END_STEP
TRANSITION FROM Back_NOK TO WaitForStart := MsgOk;
END_TRANSITION
STEP TankFront_leer:
	TankFront_leer_entry(P1);
	TankFront_leer_action(N);
	TankFront_leer_exit(P0);
END_STEP
TRANSITION FROM TankFront_leer TO WaitForStart := MsgOk;
END_TRANSITION
STEP TankBack_leer:
	TankBack_leer_entry(P1);
	TankBack_leer_action(N);
	TankBack_leer_exit(P0);
END_STEP
TRANSITION FROM TankBack_leer TO WaitForStart := MsgOk;
END_TRANSITION
STEP ErrFront:
	ErrFront_entry(P1);
	ErrFront_action(N);
	ErrFront_exit(P0);
END_STEP
TRANSITION FROM ErrFront TO WaitForStart := MsgOk;
END_TRANSITION
STEP ErrBack:
	ErrBack_entry(P1);
	ErrBack_action(N);
	ErrBack_exit(P0);
END_STEP
TRANSITION FROM ErrBack TO WaitForStart := MsgOk;
END_TRANSITION
STEP FrontCam_bb:
END_STEP
TRANSITION FROM FrontCam_bb TO FrontCam_bb_ := Frontcam_bb;
END_TRANSITION
TRANSITION FROM FrontCam_bb TO FronCam_not_bb := TRUE;
END_TRANSITION
STEP FronCam_not_bb:
	FronCam_not_bb_entry(P1);
	FronCam_not_bb_action(N);
	FronCam_not_bb_exit(P0);
END_STEP
TRANSITION FROM FronCam_not_bb TO FrontCam_bb := MsgOk;
END_TRANSITION
STEP FrontCam_bb_:
END_STEP
STEP BackCam_bb:
END_STEP
TRANSITION FROM BackCam_bb TO BackCam_bb_ := Backcam_bb;
END_TRANSITION
TRANSITION FROM BackCam_bb TO BackCam_not_bb := TRUE;
END_TRANSITION
STEP BackCam_not_bb:
	BackCam_not_bb_entry(P1);
	BackCam_not_bb_action(N);
	BackCam_not_bb_exit(P0);
END_STEP
TRANSITION FROM BackCam_not_bb TO BackCam_bb := MsgOk;
END_TRANSITION
STEP BackCam_bb_:
END_STEP
TRANSITION FROM (FrontCam_bb_, BackCam_bb_) TO (mitte_zu, hinten_auf) := Vereinzler_frei;
END_TRANSITION
TRANSITION FROM (FrontCam_bb_, BackCam_bb_) TO Delay____ := TRUE;
END_TRANSITION
STEP mitte_zu:
	mitte_zu_action(N);
END_STEP
STEP hinten_auf:
	hinten_auf_action(N);
END_STEP
TRANSITION FROM (mitte_zu, hinten_auf) TO Delay____ := StateOk;
END_TRANSITION
STEP Delay____: (* min time t#200ms; t#200ms *)
END_STEP
TRANSITION FROM Delay____ TO hinten_zu := TRUE;
END_TRANSITION
STEP hinten_zu:
	hinten_zu_action(N);
END_STEP
TRANSITION FROM hinten_zu TO Print_Cam_free := StateOk;
END_TRANSITION
STEP Print_Cam_free:
END_STEP
TRANSITION FROM Print_Cam_free TO (vorne_zu, mitte_auf) := Print_Cam_free;
END_TRANSITION
TRANSITION FROM Print_Cam_free TO Robo_free := Cam_full;
END_TRANSITION
STEP vorne_zu:
	vorne_zu_action(N);
	vorne_zu_exit(P0);
END_STEP
STEP mitte_auf:
	mitte_auf_action(N);
END_STEP
TRANSITION FROM (vorne_zu, mitte_auf) TO Iso_on_CamPos := StateOk;
END_TRANSITION
STEP Iso_on_CamPos:
END_STEP
TRANSITION FROM Iso_on_CamPos TO Delay_onCam := Iso_on_CamPos;
END_TRANSITION
STEP Delay_onCam: (* min time t#500ms; t#500ms *)
END_STEP
TRANSITION FROM Delay_onCam TO (Front_Cam_aktiv, mitte_zu_) := TRUE;
END_TRANSITION
STEP Front_Cam_aktiv:
	Front_Cam_aktiv_exit(P0);
END_STEP
TRANSITION FROM Front_Cam_aktiv TO Start_Front_Cam := aktiv;
END_TRANSITION
TRANSITION FROM Front_Cam_aktiv TO Print_Front_OK := TRUE;
END_TRANSITION
STEP Start_Front_Cam:
	Start_Front_Cam_action(N);
END_STEP
TRANSITION FROM Start_Front_Cam TO Delay_Front_Cam := Busy;
END_TRANSITION
STEP Delay_Front_Cam: (* min time t#500ms; t#500ms *)
	Delay_Front_Cam_entry(P1);
END_STEP
TRANSITION FROM Delay_Front_Cam TO Verarbeitet_FrontCam := Done;
END_TRANSITION
TRANSITION FROM Delay_Front_Cam TO Print_Front_OK := CamNotAktiv;
END_TRANSITION
TRANSITION FROM Delay_Front_Cam TO Start_Front_Cam := CamDone;
END_TRANSITION
STEP Verarbeitet_FrontCam:
	Verarbeitet_FrontCam_entry(P1);
	Verarbeitet_FrontCam_exit(P0);
END_STEP
TRANSITION FROM Verarbeitet_FrontCam TO Back_Cam_aktiv := TRUE;
END_TRANSITION
STEP Print_Front_OK:
	Print_Front_OK_exit(P0);
END_STEP
TRANSITION FROM Print_Front_OK TO Back_Cam_aktiv := TRUE;
END_TRANSITION
STEP Back_Cam_aktiv:
	Back_Cam_aktiv_exit(P0);
END_STEP
TRANSITION FROM Back_Cam_aktiv TO Start_Back_Cam := aktiv;
END_TRANSITION
TRANSITION FROM Back_Cam_aktiv TO Print_Back_OK := TRUE;
END_TRANSITION
STEP Start_Back_Cam:
	Start_Back_Cam_action(N);
END_STEP
TRANSITION FROM Start_Back_Cam TO Delay_Back_Cam := Busy;
END_TRANSITION
STEP Delay_Back_Cam: (* min time t#500ms; t#500ms *)
	Delay_Back_Cam_entry(P1);
END_STEP
TRANSITION FROM Delay_Back_Cam TO Verarbeitet_BackCam := Done;
END_TRANSITION
TRANSITION FROM Delay_Back_Cam TO Print_Back_OK := CamNotAktiv;
END_TRANSITION
TRANSITION FROM Delay_Back_Cam TO Start_Back_Cam := CamDone;
END_TRANSITION
STEP Verarbeitet_BackCam:
	Verarbeitet_BackCam_entry(P1);
	Verarbeitet_BackCam_exit(P0);
END_STEP
TRANSITION FROM Verarbeitet_BackCam TO Zylinder_2_zu := TRUE;
END_TRANSITION
STEP Print_Back_OK:
	Print_Back_OK_exit(P0);
END_STEP
TRANSITION FROM Print_Back_OK TO Zylinder_2_zu := TRUE;
END_TRANSITION
STEP Zylinder_2_zu:
	Zylinder_2_zu_action(N);
END_STEP
TRANSITION FROM Zylinder_2_zu TO Zylinder_1_auf := StateOk;
END_TRANSITION
STEP Zylinder_1_auf:
	Zylinder_1_auf_action(N);
END_STEP
TRANSITION FROM Zylinder_1_auf TO Iso_on_CamPos_2 := StateOk;
END_TRANSITION
STEP Iso_on_CamPos_2:
END_STEP
TRANSITION FROM Iso_on_CamPos_2 TO Front_Cam_aktiv__ := Iso_on_CamPos_2;
END_TRANSITION
STEP Front_Cam_aktiv__:
	Front_Cam_aktiv___exit(P0);
END_STEP
TRANSITION FROM Front_Cam_aktiv__ TO Start_Front_Cam__ := aktiv;
END_TRANSITION
TRANSITION FROM Front_Cam_aktiv__ TO Print_Front_OK__ := TRUE;
END_TRANSITION
STEP Start_Front_Cam__:
	Start_Front_Cam___action(N);
END_STEP
TRANSITION FROM Start_Front_Cam__ TO Delay_Front_Cam__ := Busy;
END_TRANSITION
STEP Delay_Front_Cam__: (* min time t#500ms; t#500ms *)
	Delay_Front_Cam___entry(P1);
END_STEP
TRANSITION FROM Delay_Front_Cam__ TO Verarbeitet_FrontCam__ := Done;
END_TRANSITION
TRANSITION FROM Delay_Front_Cam__ TO Print_Front_OK__ := CamNotAktiv;
END_TRANSITION
TRANSITION FROM Delay_Front_Cam__ TO Start_Front_Cam__ := CamDone;
END_TRANSITION
STEP Verarbeitet_FrontCam__:
	Verarbeitet_FrontCam___entry(P1);
	Verarbeitet_FrontCam___exit(P0);
END_STEP
TRANSITION FROM Verarbeitet_FrontCam__ TO Back_Cam_aktiv__ := TRUE;
END_TRANSITION
STEP Print_Front_OK__:
	Print_Front_OK___exit(P0);
END_STEP
TRANSITION FROM Print_Front_OK__ TO Back_Cam_aktiv__ := TRUE;
END_TRANSITION
STEP Back_Cam_aktiv__:
	Back_Cam_aktiv___exit(P0);
END_STEP
TRANSITION FROM Back_Cam_aktiv__ TO Start_Back_Cam__ := aktiv;
END_TRANSITION
TRANSITION FROM Back_Cam_aktiv__ TO Print_Back_OK__ := TRUE;
END_TRANSITION
STEP Start_Back_Cam__:
	Start_Back_Cam___action(N);
END_STEP
TRANSITION FROM Start_Back_Cam__ TO Delay_Back_Cam__ := Busy;
END_TRANSITION
STEP Delay_Back_Cam__: (* min time t#500ms; t#500ms *)
	Delay_Back_Cam___entry(P1);
END_STEP
TRANSITION FROM Delay_Back_Cam__ TO Verarbeitet_BackCam__ := Done;
END_TRANSITION
TRANSITION FROM Delay_Back_Cam__ TO Print_Back_OK__ := CamNotAktiv;
END_TRANSITION
TRANSITION FROM Delay_Back_Cam__ TO Start_Back_Cam__ := CamDone;
END_TRANSITION
STEP Verarbeitet_BackCam__:
	Verarbeitet_BackCam___entry(P1);
	Verarbeitet_BackCam___exit(P0);
END_STEP
TRANSITION FROM Verarbeitet_BackCam__ TO Zylinder_3_zu := TRUE;
END_TRANSITION
STEP Print_Back_OK__:
	Print_Back_OK___exit(P0);
END_STEP
TRANSITION FROM Print_Back_OK__ TO Zylinder_3_zu := TRUE;
END_TRANSITION
STEP Zylinder_3_zu:
	Zylinder_3_zu_action(N);
END_STEP
TRANSITION FROM Zylinder_3_zu TO Zylinder_2_auf := StateOk;
END_TRANSITION
STEP Zylinder_2_auf:
	Zylinder_2_auf_action(N);
END_STEP
TRANSITION FROM Zylinder_2_auf TO Iso_on_CamPos_3 := StateOk;
END_TRANSITION
STEP Iso_on_CamPos_3:
END_STEP
TRANSITION FROM Iso_on_CamPos_3 TO Front_Cam_aktiv_ := Iso_on_CamPos_2;
END_TRANSITION
STEP Front_Cam_aktiv_:
	Front_Cam_aktiv__exit(P0);
END_STEP
TRANSITION FROM Front_Cam_aktiv_ TO Start_Front_Cam_ := aktiv;
END_TRANSITION
TRANSITION FROM Front_Cam_aktiv_ TO Print_Front_OK_ := TRUE;
END_TRANSITION
STEP Start_Front_Cam_:
	Start_Front_Cam__action(N);
END_STEP
TRANSITION FROM Start_Front_Cam_ TO Delay_Front_Cam_ := Busy;
END_TRANSITION
STEP Delay_Front_Cam_: (* min time t#500ms; t#500ms *)
	Delay_Front_Cam__entry(P1);
END_STEP
TRANSITION FROM Delay_Front_Cam_ TO Verarbeitet_FrontCam_ := Done;
END_TRANSITION
TRANSITION FROM Delay_Front_Cam_ TO Print_Front_OK_ := CamNotAktiv;
END_TRANSITION
TRANSITION FROM Delay_Front_Cam_ TO Start_Front_Cam_ := CamDone;
END_TRANSITION
STEP Verarbeitet_FrontCam_:
	Verarbeitet_FrontCam__entry(P1);
	Verarbeitet_FrontCam__exit(P0);
END_STEP
TRANSITION FROM Verarbeitet_FrontCam_ TO Back_Cam_aktiv_ := TRUE;
END_TRANSITION
STEP Print_Front_OK_:
	Print_Front_OK__exit(P0);
END_STEP
TRANSITION FROM Print_Front_OK_ TO Back_Cam_aktiv_ := TRUE;
END_TRANSITION
STEP Back_Cam_aktiv_:
	Back_Cam_aktiv__exit(P0);
END_STEP
TRANSITION FROM Back_Cam_aktiv_ TO Start_Back_Cam_ := aktiv;
END_TRANSITION
TRANSITION FROM Back_Cam_aktiv_ TO Print_Back_OK_ := TRUE;
END_TRANSITION
STEP Start_Back_Cam_:
	Start_Back_Cam__action(N);
END_STEP
TRANSITION FROM Start_Back_Cam_ TO Delay_Back_Cam_ := Busy;
END_TRANSITION
STEP Delay_Back_Cam_: (* min time t#500ms; t#500ms *)
	Delay_Back_Cam__entry(P1);
END_STEP
TRANSITION FROM Delay_Back_Cam_ TO Verarbeitet_BackCam_ := Done;
END_TRANSITION
TRANSITION FROM Delay_Back_Cam_ TO Print_Back_OK_ := CamNotAktiv;
END_TRANSITION
TRANSITION FROM Delay_Back_Cam_ TO Start_Back_Cam_ := CamDone;
END_TRANSITION
STEP Verarbeitet_BackCam_:
	Verarbeitet_BackCam__entry(P1);
	Verarbeitet_BackCam__exit(P0);
END_STEP
TRANSITION FROM Verarbeitet_BackCam_ TO Step54 := TRUE;
END_TRANSITION
STEP Print_Back_OK_:
	Print_Back_OK__exit(P0);
END_STEP
TRANSITION FROM Print_Back_OK_ TO Step54 := TRUE;
END_TRANSITION
STEP Step54:
END_STEP
STEP mitte_zu_:
	mitte_zu__action(N);
END_STEP
TRANSITION FROM mitte_zu_ TO hinten_auf_ := StateOk;
END_TRANSITION
STEP hinten_auf_:
	hinten_auf__action(N);
END_STEP
TRANSITION FROM hinten_auf_ TO Step43 := StateOk;
END_TRANSITION
STEP Step43:
END_STEP
TRANSITION FROM (Step54, Step43) TO ResetNokCounter := TRUE;
END_TRANSITION
STEP ResetNokCounter:
	ResetNokCounter_entry(P1);
END_STEP
TRANSITION FROM ResetNokCounter TO CheckCounter := TRUE;
END_TRANSITION
STEP CheckCounter:
	CheckCounter_entry(P1);
END_STEP
TRANSITION FROM CheckCounter TO Robo_free := CounterOK;
END_TRANSITION
TRANSITION FROM CheckCounter TO Msg_Cam := Nok_Cont;
END_TRANSITION
TRANSITION FROM CheckCounter TO Msg_Cam_Percent := Nok_Percent;
END_TRANSITION
STEP Msg_Cam:
	Msg_Cam_entry(P1);
	Msg_Cam_action(N);
	Msg_Cam_exit(P0);
END_STEP
TRANSITION FROM Msg_Cam TO Counter_Reset := MsgOK;
END_TRANSITION
STEP Counter_Reset:
	Counter_Reset_entry(P1);
END_STEP
TRANSITION FROM Counter_Reset TO Robo_free := TRUE;
END_TRANSITION
STEP Msg_Cam_Percent:
	Msg_Cam_Percent_entry(P1);
	Msg_Cam_Percent_action(N);
	Msg_Cam_Percent_exit(P0);
END_STEP
TRANSITION FROM Msg_Cam_Percent TO Counter_Reset := MsgOK;
END_TRANSITION
STEP Robo_free:
END_STEP
TRANSITION FROM Robo_free TO Zylinder_3_auf_ := free;
END_TRANSITION
TRANSITION FROM Robo_free TO SeqEnd := TRUE;
END_TRANSITION
STEP Zylinder_3_auf_:
	Zylinder_3_auf__action(N);
	Zylinder_3_auf__exit(P0);
END_STEP
TRANSITION FROM Zylinder_3_auf_ TO Delay_ := StateOk;
END_TRANSITION
STEP Delay_: (* min time t#500ms; t#500ms *)
END_STEP
TRANSITION FROM Delay_ TO Zylinder_1_zu_ := TRUE;
END_TRANSITION
STEP Zylinder_1_zu_:
	Zylinder_1_zu__action(N);
END_STEP
TRANSITION FROM Zylinder_1_zu_ TO SeqEnd := StateOk;
END_TRANSITION
STEP SeqEnd: (* -> WAIT *)
	SeqEnd_action(N);
END_STEP
TRANSITION FROM SeqEnd TO WaitForStart := TRUE;
END_TRANSITION

ACTION Init_action:
Start:=FALSE;
State:=STATE_WAIT;
MsgOK:=FALSE;
MsgCancel:=FALSE;
SFCRun:=FALSE;
Result160pol:=RESULT_NON;
NokCounter:=0;

ST03_8_80_A1.b_start := FALSE;
ST03_8_85_A1.b_start := FALSE;

ST03_8_90_A1.st_ctrl_in.b_start := FALSE;
ST03_8_95_A1.st_ctrl_in.b_start := FALSE;
END_ACTION

ACTION WaitForStart_entry:
;
END_ACTION

ACTION WaitForStart_action:
IF 	Start   THEN
	State:=STATE_RUN;
	SFCTimeStart:=TIME();
	Start:=FALSE;
ELSE
	State:=STATE_WAIT;
	MsgOK:=FALSE;
	MsgCancel:=FALSE;
	SFCRun:=FALSE;
END_IF
END_ACTION

ACTION TDA_Luft_NOK_entry:
MessageHandler.ClearMessageLines(sVisu:=Visu.Message);
END_ACTION

ACTION TDA_Luft_NOK_action:
MessageHandler.Msg.ID:='PM103';
MessageHandler.Msg.Name:='Tintenstrahldrucker Druckschalter';
MessageHandler.Msg.Text:='ST02 Druckschalter Wartungseinheit Hauptluft min.6 bar';
MessageHandler.Msg.Color:=Color.red;
MessageHandler.Msg.Station:=1;


MessageHandler(
	Prio:=2, 							(*1=highest, .. , 4=lowest*)
	Btn1Addr:=ADR(MsgOk),			(*Address of Button1 , if Zero then Button is unvisible*)
	Btn2Addr:=,						(*Address of Button2 , if Zero then Button is unvisible*)
	sVisu:=Visu.Message);
END_ACTION

ACTION TDA_Luft_NOK_exit:
MsgOk:=FALSE;
MsgCancel:=FALSE;
END_ACTION

ACTION LampsPrint_action:
(*Signalsäule Tintenstrahldrucker schalten, nur bei SGM-3621*)

(*Signalsäuele Bedruckung RD Sammelstörung*)
ST03_H7.SetSignalHigh:= FALSE;
ST03_H7.SetSignalLow:= TRUE;
(*Signalsäule Bedruckung GR Bedruckung IO*)
ST03_H6.SetSignalHigh:= TRUE;
ST03_H6.SetSignalLow:= FALSE;
END_ACTION

ACTION Front_NOK_entry:
MessageHandler.ClearMessageLines(sVisu:=Visu.Message);
END_ACTION

ACTION Front_NOK_action:
MessageHandler.Msg.ID:='PM104';
MessageHandler.Msg.Name:=ST03_70U3_1.sInit.Description;
MessageHandler.Msg.Text:='Drucker Front nicht betriebsbereit';
MessageHandler.Msg.Color:=Color.red;
MessageHandler.Msg.Station:=1;


MessageHandler(
	Prio:=2, 							(*1=highest, .. , 4=lowest*)
	Btn1Addr:=ADR(MsgOk),			(*Address of Button1 , if Zero then Button is unvisible*)
	Btn2Addr:=,						(*Address of Button2 , if Zero then Button is unvisible*)
	sVisu:=Visu.Message);
END_ACTION

ACTION Front_NOK_exit:
MsgOk:=FALSE;
MsgCancel:=FALSE;
END_ACTION

ACTION Back_NOK_entry:
MessageHandler.ClearMessageLines(sVisu:=Visu.Message);
END_ACTION

ACTION Back_NOK_action:
MessageHandler.Msg.ID:='PM105';
MessageHandler.Msg.Name:=ST03_71U3_1.sInit.Description;
MessageHandler.Msg.Text:='Drucker Rückseite nicht betriebsbereit';
MessageHandler.Msg.Color:=Color.red;
MessageHandler.Msg.Station:=1;


MessageHandler(
	Prio:=2, 							(*1=highest, .. , 4=lowest*)
	Btn1Addr:=ADR(MsgOk),			(*Address of Button1 , if Zero then Button is unvisible*)
	Btn2Addr:=,						(*Address of Button2 , if Zero then Button is unvisible*)
	sVisu:=Visu.Message);
END_ACTION

ACTION Back_NOK_exit:
MsgOk:=FALSE;
MsgCancel:=FALSE;
END_ACTION

ACTION TankFront_leer_entry:
MessageHandler.ClearMessageLines(sVisu:=Visu.Message);
END_ACTION

ACTION TankFront_leer_action:
MessageHandler.Msg.ID:='PM106';
MessageHandler.Msg.Name:=ST03_70U3_2.sInit.Description;
MessageHandler.Msg.Text:='Tank Drucker Frontseite leer';
MessageHandler.Msg.Color:=Color.red;
MessageHandler.Msg.Station:=1;


MessageHandler(
	Prio:=2, 							(*1=highest, .. , 4=lowest*)
	Btn1Addr:=ADR(MsgOk),			(*Address of Button1 , if Zero then Button is unvisible*)
	Btn2Addr:=,						(*Address of Button2 , if Zero then Button is unvisible*)
	sVisu:=Visu.Message);
END_ACTION

ACTION TankFront_leer_exit:
MsgOk:=FALSE;
MsgCancel:=FALSE;
END_ACTION

ACTION TankBack_leer_entry:
MessageHandler.ClearMessageLines(sVisu:=Visu.Message);
END_ACTION

ACTION TankBack_leer_action:
MessageHandler.Msg.ID:='PM107';
MessageHandler.Msg.Name:=ST03_71U3_2.sInit.Description;
MessageHandler.Msg.Text:='Tank Drucker Rückseite leer';
MessageHandler.Msg.Color:=Color.red;
MessageHandler.Msg.Station:=1;


MessageHandler(
	Prio:=2, 							(*1=highest, .. , 4=lowest*)
	Btn1Addr:=ADR(MsgOk),			(*Address of Button1 , if Zero then Button is unvisible*)
	Btn2Addr:=,						(*Address of Button2 , if Zero then Button is unvisible*)
	sVisu:=Visu.Message);
END_ACTION

ACTION TankBack_leer_exit:
MsgOk:=FALSE;
MsgCancel:=FALSE;
END_ACTION

ACTION ErrFront_entry:
MessageHandler.ClearMessageLines(sVisu:=Visu.Message);
(*Signalsäuele Bedruckung RD Sammelstörung*)
ST03_H7.SetSignalHigh:= TRUE;
ST03_H7.SetSignalLow:= FALSE;
(*Signalsäule Bedruckung GR Bedruckung IO*)
ST03_H6.SetSignalHigh:= FALSE;
ST03_H6.SetSignalLow:= TRUE;
END_ACTION

ACTION ErrFront_action:
MessageHandler.Msg.ID:='PM108';
MessageHandler.Msg.Name:=ST03_70U3_3.sInit.Description;
MessageHandler.Msg.Text:='Störung Drucker Frontseite ';
MessageHandler.Msg.Color:=Color.red;
MessageHandler.Msg.Station:=1;


MessageHandler(
	Prio:=2, 							(*1=highest, .. , 4=lowest*)
	Btn1Addr:=ADR(MsgOk),			(*Address of Button1 , if Zero then Button is unvisible*)
	Btn2Addr:=,						(*Address of Button2 , if Zero then Button is unvisible*)
	sVisu:=Visu.Message);
END_ACTION

ACTION ErrFront_exit:
MsgOk:=FALSE;
MsgCancel:=FALSE;
(*Signalsäuele Bedruckung RD Sammelstörung*)
ST03_H7.SetSignalHigh:= FALSE;
ST03_H7.SetSignalLow:= TRUE;
(*Signalsäule Bedruckung GR Bedruckung IO*)
ST03_H6.SetSignalHigh:= TRUE;
ST03_H6.SetSignalLow:= FALSE;
END_ACTION

ACTION ErrBack_entry:
MessageHandler.ClearMessageLines(sVisu:=Visu.Message);
(*Signalsäuele Bedruckung RD Sammelstörung*)
ST03_H7.SetSignalHigh:= TRUE;
ST03_H7.SetSignalLow:= FALSE;
(*Signalsäule Bedruckung GR Bedruckung IO*)
ST03_H6.SetSignalHigh:= FALSE;
ST03_H6.SetSignalLow:= TRUE;
END_ACTION

ACTION ErrBack_action:
MessageHandler.Msg.ID:='PM109';
MessageHandler.Msg.Name:=ST03_71U3_3.sInit.Description;
MessageHandler.Msg.Text:='Störung Drucker Rückseite';
MessageHandler.Msg.Color:=Color.red;
MessageHandler.Msg.Station:=1;


MessageHandler(
	Prio:=2, 							(*1=highest, .. , 4=lowest*)
	Btn1Addr:=ADR(MsgOk),			(*Address of Button1 , if Zero then Button is unvisible*)
	Btn2Addr:=,						(*Address of Button2 , if Zero then Button is unvisible*)
	sVisu:=Visu.Message);
END_ACTION

ACTION ErrBack_exit:
MsgOk:=FALSE;
MsgCancel:=FALSE;
(*Signalsäuele Bedruckung RD Sammelstörung*)
ST03_H7.SetSignalHigh:= FALSE;
ST03_H7.SetSignalLow:= TRUE;
(*Signalsäule Bedruckung GR Bedruckung IO*)
ST03_H6.SetSignalHigh:= TRUE;
ST03_H6.SetSignalLow:= FALSE;
END_ACTION

ACTION FronCam_not_bb_entry:
MessageHandler.ClearMessageLines(sVisu:=Visu.Message);
END_ACTION

ACTION FronCam_not_bb_action:
MessageHandler.Msg.ID:='PM110';
MessageHandler.Msg.Name:='Check Camera';
MessageHandler.Msg.Text:='Kamera Frontseite ist nicht betriebsbereit';
MessageHandler.Msg.Color:=Color.red;
MessageHandler.Msg.Station:=1;


MessageHandler(
	Prio:=2, 							(*1=highest, .. , 4=lowest*)
	Btn1Addr:=ADR(MsgOk),			(*Address of Button1 , if Zero then Button is unvisible*)
	Btn2Addr:=,						(*Address of Button2 , if Zero then Button is unvisible*)
	sVisu:=Visu.Message);
END_ACTION

ACTION FronCam_not_bb_exit:
MsgOk:=FALSE;
MsgCancel:=FALSE;
END_ACTION

ACTION BackCam_not_bb_entry:
MessageHandler.ClearMessageLines(sVisu:=Visu.Message);
END_ACTION

ACTION BackCam_not_bb_action:
MessageHandler.Msg.ID:='PM111';
MessageHandler.Msg.Name:='Check Camera';
MessageHandler.Msg.Text:='Kamera Rückseite ist nicht betriebsbereit';
MessageHandler.Msg.Color:=Color.red;
MessageHandler.Msg.Station:=1;


MessageHandler(
	Prio:=2, 							(*1=highest, .. , 4=lowest*)
	Btn1Addr:=ADR(MsgOk),			(*Address of Button1 , if Zero then Button is unvisible*)
	Btn2Addr:=,						(*Address of Button2 , if Zero then Button is unvisible*)
	sVisu:=Visu.Message);
END_ACTION

ACTION BackCam_not_bb_exit:
MsgOk:=FALSE;
MsgCancel:=FALSE;
END_ACTION

ACTION mitte_zu_action:
ST03_422_Y64_6.MoveInit:=TRUE;	(* Förderband  Stopper Vereinzler AST/GST *)
END_ACTION

ACTION hinten_auf_action:
ST03_422_Y64_5.MoveInit:=TRUE;
END_ACTION

ACTION hinten_zu_action:
ST03_422_Y64_5.MoveWork:=TRUE;	(* Förderband  Stopper Vereinzler AST/GST *)
END_ACTION

ACTION vorne_zu_action:
ST03_422_Y64_7.MoveWork:=TRUE;
END_ACTION

ACTION vorne_zu_exit:
CamResult:=0;
END_ACTION

ACTION mitte_auf_action:
ST03_422_Y64_6.MoveWork :=TRUE;
END_ACTION

ACTION Front_Cam_aktiv_exit:
RepeatCounter:=0;
CamResult:=0;
CamResult2:=0;
CamResult3:=0;
END_ACTION

ACTION Start_Front_Cam_action:
IF NOT MP.ST02.SensopartEthernet THEN
	ST03_8_80_A1.i16_job := 1;		 (*Sensopart Kamera Frontseite*)
	ST03_8_80_A1.b_start := TRUE;
ELSE
	ST03_8_90_A1.JobNo := 1;
	ST03_8_90_A1.st_ctrl_in.b_start := TRUE;
END_IF
END_ACTION

ACTION Delay_Front_Cam_entry:
IF NOT MP.ST02.SensopartEthernet THEN
	ST03_8_80_A1.b_start := FALSE;	 (*Sensopart Kamera Frontseite*)
ELSE
	ST03_8_90_A1.st_ctrl_in.b_start := FALSE;
END_IF

RepeatCounter:=RepeatCounter+1;
END_ACTION

ACTION Verarbeitet_FrontCam_entry:
IF NOT MP.ST02.SensopartEthernet THEN
	IF 	MP.ST03.FrontCamOn THEN
		IF	ST03_8_80_A1.Ergebnis_IO AND	  (*Sensopart Kamera  links*)
			NOT ST03_8_80_A1.Ergebnis_NIO THEN
			CamResult:=1;	(*   0 = noch kein Bild gemacht*)
						(*   1 =  Frontseite OK*)
						(*  11 = Frontseite und Rückseite OK*)
						(*  99 = Teil ist NOK	*)
		ELSE
			CamResult:=9;	(*   0 = noch kein Bild gemacht*)
						(*   1 =  Frontseite OK*)
						(*  11 = Frontseite und Rückseite OK*)
						(*  99 = Teil ist NOK	*)
		END_IF

	ELSE
		CamResult:=1;		(*   1 =  Frontseite OK*)
	END_IF
ELSE
		IF 	MP.ST03.FrontCamOn THEN
		IF	ST03_8_90_A1.b_Kam_Pruef_IO AND	  (*Sensopart Kamera links*)
			NOT ST03_8_90_A1.b_Kam_Pruef_NIO THEN
			CamResult:=1;	(*   0 = noch kein Bild gemacht*)
						(*   1 =  Frontseite OK*)
						(*  11 = Frontseite und Rückseite OK*)
						(*  99 = Teil ist NOK	*)
		ELSE
			CamResult:=9;	(*   0 = noch kein Bild gemacht*)
						(*   1 =  Frontseite OK*)
						(*  11 = Frontseite und Rückseite OK*)
						(*  99 = Teil ist NOK	*)
		END_IF
	
	ELSE
		CamResult:=1;		(*   1 =  Frontseite OK*)
	END_IF
END_IF
	RepeatCounter:=RepeatCounter+1;
END_ACTION

ACTION Verarbeitet_FrontCam_exit:
IF CamResult = 9 THEN
	NokCounter1li := NokCounter1li + 1;
END_IF
END_ACTION

ACTION Print_Front_OK_exit:
CamResult:=1;	(*   0 = noch kein Bild gemacht*)
			(*   1 =  Frontseite OK*)
			(*  11 = Frontseite und Rückseite OK*)
			(*  99 = Teil ist NOK	*)
END_ACTION

ACTION Back_Cam_aktiv_exit:
RepeatCounter:=0;
END_ACTION

ACTION Start_Back_Cam_action:
IF NOT MP.ST02.SensopartEthernet THEN
	ST03_8_85_A1.i16_job := 1;		 (*Sensopart Kamera rechts*)
	ST03_8_85_A1.b_start := TRUE;
ELSE
	ST03_8_95_A1.JobNo := 1;		(*Sensopart Kamera Ethernet rechts *)
	ST03_8_95_A1.st_ctrl_in.b_start := TRUE;
END_IF
END_ACTION

ACTION Delay_Back_Cam_entry:
IF NOT MP.ST02.SensopartEthernet THEN
	ST03_8_85_A1.b_start := FALSE;	 (*Sensopart Kamera rechts*)
ELSE
	ST03_8_95_A1.st_ctrl_in.b_start := FALSE;	(*Sensopart Kamera Ethernet rechts *)
END_IF

RepeatCounter:=RepeatCounter+1;
END_ACTION

ACTION Verarbeitet_BackCam_entry:
IF NOT MP.ST02.SensopartEthernet THEN
	IF 	MP.ST03.BackCamOn THEN
		IF	ST03_8_85_A1.Ergebnis_IO AND	  (*Sensopart Kamera rechts*)
			NOT ST03_8_85_A1.Ergebnis_NIO THEN
			CamResult:=CamResult+10;	(*   0 = noch kein Bild gemacht*)
							(*   1 =  Frontseite OK*)
							(*  11 = Frontseite und Rückseite OK*)
							(*  99 = Teil ist NOK	*)
		ELSE
			CamResult:=99;		(*   0 = noch kein Bild gemacht*)
							(*   1 =  Frontseite OK*)
							(*  11 = Frontseite und Rückseite OK*)
							(*  99 = Teil ist NOK	*)
		END_IF
	
	ELSE
		CamResult:=CamResult+10;		(*   1 =  Frontseite OK*)
	END_IF

ELSE
		IF 	MP.ST03.FrontCamOn THEN
		IF	ST03_8_95_A1.b_Kam_Pruef_IO AND	 (*Sensopart Kamera Ethernet rechts *)
			NOT ST03_8_95_A1.b_Kam_Pruef_NIO THEN
			CamResult:=CamResult+10;	(*   0 = noch kein Bild gemacht*)
						(*   1 =  Frontseite OK*)
						(*  11 = Frontseite und Rückseite OK*)
						(*  99 = Teil ist NOK	*)
		ELSE
			CamResult:=CamResult + 90;	(*   0 = noch kein Bild gemacht*)
						(*   1 =  Frontseite OK*)
						(*  11 = Frontseite und Rückseite OK*)
						(*  99 = Teil ist NOK	*)
		END_IF
	
	ELSE
		CamResult:=CamResult+10;		(*   1 =  Rückseite OK*)
	END_IF
END_IF
RepeatCounter:=RepeatCounter+1;
END_ACTION

ACTION Verarbeitet_BackCam_exit:
IF CamResult > 19 THEN
	NokCounter1re := NokCounter1re +1;
END_IF
END_ACTION

ACTION Print_Back_OK_exit:
CamResult:=CamResult+10;	(*   0 = noch kein Bild gemacht*)
				(*   1 =  Frontseite OK*)
				(*  11 = Frontseite und Rückseite OK*)
				(*  99 = Teil ist NOK	*)
END_ACTION

ACTION Zylinder_2_zu_action:
ST03_423_Y65_6.MoveWork := TRUE;
END_ACTION

ACTION Zylinder_1_auf_action:
ST03_422_Y64_7.MoveInit := TRUE;
END_ACTION

ACTION Front_Cam_aktiv___exit:
RepeatCounter:=0;
CamResult2:=0;
END_ACTION

ACTION Start_Front_Cam___action:
IF NOT MP.ST02.SensopartEthernet THEN
	ST03_8_80_A1.i16_job := 1;		 (*Sensopart Kamera Frontseite*)
	ST03_8_80_A1.b_start := TRUE;
ELSE
	ST03_8_90_A1.JobNo := 2;
	ST03_8_90_A1.st_ctrl_in.b_start := TRUE;
END_IF
END_ACTION

ACTION Delay_Front_Cam___entry:
IF NOT MP.ST02.SensopartEthernet THEN
	ST03_8_80_A1.b_start := FALSE;			 (*Sensopart Kamera links*)
ELSE
	ST03_8_90_A1.st_ctrl_in.b_start := FALSE;	 (*Sensopart Kamera Ethernet links *)
END_IF

RepeatCounter:=RepeatCounter+1;
END_ACTION

ACTION Verarbeitet_FrontCam___entry:
IF NOT MP.ST02.SensopartEthernet THEN
	IF 	MP.ST03.FrontCamOn THEN
		IF	ST03_8_80_A1.Ergebnis_IO AND	  (*Sensopart Kamera links*)
			NOT ST03_8_80_A1.Ergebnis_NIO THEN
			CamResult2:=1;	(*   0 = noch kein Bild gemacht*)
						(*   1 =  Frontseite OK*)
						(*  11 = Frontseite und Rückseite OK*)
						(*  99 = Teil ist NOK	*)
		ELSE
			CamResult2:=9;	(*   0 = noch kein Bild gemacht*)
						(*   1 =  Frontseite OK*)
						(*  11 = Frontseite und Rückseite OK*)
						(*  99 = Teil ist NOK	*)
		END_IF
	
	ELSE
		CamResult2:=1;		(*   1 =  Frontseite OK*)
	END_IF
ELSE
		IF 	MP.ST03.FrontCamOn THEN
		IF	ST03_8_90_A1.b_Kam_Pruef_IO AND	   (*Sensopart Kamera Ethernet links *)
			NOT ST03_8_90_A1.b_Kam_Pruef_NIO THEN
			CamResult2:=1;	(*   0 = noch kein Bild gemacht*)
						(*   1 =  Frontseite OK*)
						(*  11 = Frontseite und Rückseite OK*)
						(*  99 = Teil ist NOK	*)
		ELSE
			CamResult2:=9;	(*   0 = noch kein Bild gemacht*)
						(*   1 =  Frontseite OK*)
						(*  11 = Frontseite und Rückseite OK*)
						(*  99 = Teil ist NOK	*)
		END_IF
	
	ELSE
		CamResult2:=1;		(*   1 =  Frontseite OK*)
	END_IF
END_IF
	RepeatCounter:=RepeatCounter+1;
END_ACTION

ACTION Verarbeitet_FrontCam___exit:
IF CamResult2 = 9 THEN
	NokCounter2li := NokCounter2li +1;
END_IF
END_ACTION

ACTION Print_Front_OK___exit:
CamResult2:=1;	(*   0 = noch kein Bild gemacht*)
			(*   1 =  Frontseite OK*)
			(*  11 = Frontseite und Rückseite OK*)
			(*  99 = Teil ist NOK	*)
END_ACTION

ACTION Back_Cam_aktiv___exit:
RepeatCounter:=0;
END_ACTION

ACTION Start_Back_Cam___action:
IF NOT MP.ST02.SensopartEthernet THEN
	ST03_8_85_A1.i16_job := 1;		 (*Sensopart Kamera rechts*)
	ST03_8_85_A1.b_start := TRUE;
ELSE
	ST03_8_95_A1.JobNo := 2;		(*Sensopart Kamera Ethernet rechts *)
	ST03_8_95_A1.st_ctrl_in.b_start := TRUE;
END_IF
END_ACTION

ACTION Delay_Back_Cam___entry:
IF NOT MP.ST02.SensopartEthernet THEN
	ST03_8_85_A1.b_start := FALSE;			 (*Sensopart Kamera rechts*)
ELSE
	ST03_8_95_A1.st_ctrl_in.b_start := FALSE;	(*Sensopart Kamera Ethernet rechts *)
END_IF

RepeatCounter:=RepeatCounter+1;
END_ACTION

ACTION Verarbeitet_BackCam___entry:
IF NOT MP.ST02.SensopartEthernet THEN
	IF 	MP.ST03.BackCamOn THEN
		IF	ST03_8_85_A1.Ergebnis_IO AND	  (*Sensopart Kamera rechts*)
			NOT ST03_8_85_A1.Ergebnis_NIO THEN
			CamResult2:=CamResult2+10;	(*   0 = noch kein Bild gemacht*)
							(*   1 =  Frontseite OK*)
							(*  11 = Frontseite und Rückseite OK*)
							(*  99 = Teil ist NOK	*)
		ELSE
			CamResult2:=99;		(*   0 = noch kein Bild gemacht*)
							(*   1 =  Frontseite OK*)
							(*  11 = Frontseite und Rückseite OK*)
							(*  99 = Teil ist NOK	*)
		END_IF

	ELSE
		CamResult2:=CamResult2+10;		(*   1 =  Rückseite OK*)
	END_IF

ELSE
		IF 	MP.ST03.FrontCamOn THEN
		IF	ST03_8_95_A1.b_Kam_Pruef_IO AND	  (*Sensopart Kamera Ethernet rechts *)
			NOT ST03_8_95_A1.b_Kam_Pruef_NIO THEN
			CamResult2:=CamResult2+10;	(*   0 = noch kein Bild gemacht*)
						(*   1 =  Frontseite OK*)
						(*  11 = Frontseite und Rückseite OK*)
						(*  99 = Teil ist NOK	*)
		ELSE
			CamResult2:=CamResult2 + 90;	(*   0 = noch kein Bild gemacht*)
						(*   1 =  Frontseite OK*)
						(*  11 = Frontseite und Rückseite OK*)
						(*  99 = Teil ist NOK	*)
		END_IF

	ELSE
		CamResult2:=CamResult2+10;			(*   1 =  Rückseite OK*)
	END_IF
END_IF
RepeatCounter:=RepeatCounter+1;
END_ACTION

ACTION Verarbeitet_BackCam___exit:
IF CamResult2 > 19 THEN
	NokCounter2re := NokCounter2re +1;
END_IF
END_ACTION

ACTION Print_Back_OK___exit:
CamResult2:=CamResult2+10;	(*   0 = noch kein Bild gemacht*)
				(*   1 =  Frontseite OK*)
				(*  11 = Frontseite und Rückseite OK*)
				(*  99 = Teil ist NOK	*)
END_ACTION

ACTION Zylinder_3_zu_action:
ST03_423_Y65_7.MoveInit := TRUE;
END_ACTION

ACTION Zylinder_2_auf_action:
ST03_423_Y65_6.MoveInit := TRUE;
END_ACTION

ACTION Front_Cam_aktiv__exit:
RepeatCounter:=0;
CamResult3:=0;
END_ACTION

ACTION Start_Front_Cam__action:
IF NOT MP.ST02.SensopartEthernet THEN
	ST03_8_80_A1.i16_job := 1;		 (*Sensopart Kamera links*)
	ST03_8_80_A1.b_start := TRUE;
ELSE
	ST03_8_90_A1.JobNo := 3;		(*Sensopart Kamera Ethernet links *)
	ST03_8_90_A1.st_ctrl_in.b_start := TRUE;
END_IF
END_ACTION

ACTION Delay_Front_Cam__entry:
IF NOT MP.ST02.SensopartEthernet THEN
	ST03_8_80_A1.b_start := FALSE;	 (*Sensopart Kamera links*)
ELSE
	ST03_8_90_A1.st_ctrl_in.b_start := FALSE;	(*Sensopart Kamera Ethernet links *)
END_IF

RepeatCounter:=RepeatCounter+1;
END_ACTION

ACTION Verarbeitet_FrontCam__entry:
IF NOT MP.ST02.SensopartEthernet THEN
	IF 	MP.ST03.FrontCamOn THEN
		IF	ST03_8_80_A1.Ergebnis_IO AND	  (*Sensopart Kamera links*)
			NOT ST03_8_80_A1.Ergebnis_NIO THEN
			CamResult3:=1;	(*   0 = noch kein Bild gemacht*)
						(*   1 =  Frontseite OK*)
						(*  11 = Frontseite und Rückseite OK*)
						(*  99 = Teil ist NOK	*)
		ELSE
			CamResult3:=9;	(*   0 = noch kein Bild gemacht*)
						(*   1 =  Frontseite OK*)
						(*  11 = Frontseite und Rückseite OK*)
						(*  99 = Teil ist NOK	*)
		END_IF

	ELSE
		CamResult3:=1;		(*   1 =  Frontseite OK*)
	END_IF
ELSE
		IF 	MP.ST03.FrontCamOn THEN
		IF	ST03_8_90_A1.b_Kam_Pruef_IO AND	 (*Sensopart Kamera Ethernet links *)
			NOT ST03_8_90_A1.b_Kam_Pruef_NIO THEN
			CamResult3:=1;	(*   0 = noch kein Bild gemacht*)
						(*   1 =  Frontseite OK*)
						(*  11 = Frontseite und Rückseite OK*)
						(*  99 = Teil ist NOK	*)
		ELSE
			CamResult3:=9;	(*   0 = noch kein Bild gemacht*)
						(*   1 =  Frontseite OK*)
						(*  11 = Frontseite und Rückseite OK*)
						(*  99 = Teil ist NOK	*)
		END_IF

	ELSE
		CamResult3:=1;		(*   1 =  Frontseite OK*)
	END_IF
END_IF
	RepeatCounter:=RepeatCounter+1;
END_ACTION

ACTION Verarbeitet_FrontCam__exit:
IF CamResult3 = 9 THEN
	NokCounter3li := NokCounter3li +1;
END_IF
END_ACTION

ACTION Print_Front_OK__exit:
CamResult3:=1;	(*   0 = noch kein Bild gemacht*)
			(*   1 =  Frontseite OK*)
			(*  11 = Frontseite und Rückseite OK*)
			(*  99 = Teil ist NOK	*)
END_ACTION

ACTION Back_Cam_aktiv__exit:
RepeatCounter:=0;
END_ACTION

ACTION Start_Back_Cam__action:
IF NOT MP.ST02.SensopartEthernet THEN
	ST03_8_85_A1.i16_job := 1;		 (*Sensopart Kamera rechts*)
	ST03_8_85_A1.b_start := TRUE;
ELSE
	ST03_8_95_A1.JobNo := 3;		(*Sensopart Kamera Ethernet rechts *)
	ST03_8_95_A1.st_ctrl_in.b_start := TRUE;
END_IF
END_ACTION

ACTION Delay_Back_Cam__entry:
IF NOT MP.ST02.SensopartEthernet THEN
	ST03_8_85_A1.b_start := FALSE;	 (*Sensopart Kamera rechts*)
ELSE
	ST03_8_95_A1.st_ctrl_in.b_start := FALSE;	(*Sensopart Kamera Ethernet rechts *)
END_IF

RepeatCounter:=RepeatCounter+1;
END_ACTION

ACTION Verarbeitet_BackCam__entry:
IF NOT MP.ST02.SensopartEthernet THEN
	IF 	MP.ST03.BackCamOn THEN
		IF	ST03_8_85_A1.Ergebnis_IO AND	  (*Sensopart Kamera rechts*)
			NOT ST03_8_85_A1.Ergebnis_NIO THEN
			CamResult3:=CamResult3+10;	(*   0 = noch kein Bild gemacht*)
							(*   1 =  Frontseite OK*)
							(*  11 = Frontseite und Rückseite OK*)
							(*  99 = Teil ist NOK	*)
		ELSE
			CamResult3:= 99;		(*   0 = noch kein Bild gemacht*)
							(*   1 =  Frontseite OK*)
							(*  11 = Frontseite und Rückseite OK*)
							(*  99 = Teil ist NOK	*)
		END_IF
	
	ELSE
		CamResult3:=CamResult3+10;		(*   1 =  Frontseite OK*)
	END_IF

ELSE
		IF 	MP.ST03.BackCamOn THEN
		IF	ST03_8_95_A1.b_Kam_Pruef_IO AND	 (*Sensopart Kamera Ethernet rechts *)
			NOT ST03_8_95_A1.b_Kam_Pruef_NIO THEN
			CamResult3:=CamResult3+10;	(*   0 = noch kein Bild gemacht*)
						(*   1 =  Frontseite OK*)
						(*  11 = Frontseite und Rückseite OK*)
						(*  99 = Teil ist NOK	*)
		ELSE
			CamResult3:=CamResult3 + 90;	(*   0 = noch kein Bild gemacht*)
						(*   1 =  Frontseite OK*)
						(*  11 = Frontseite und Rückseite OK*)
						(*  99 = Teil ist NOK	*)
		END_IF
	
	ELSE
		CamResult3:=CamResult3+10;		(*   1 =  Rückseite OK*)
	END_IF
END_IF
RepeatCounter:=RepeatCounter+1;
END_ACTION

ACTION Verarbeitet_BackCam__exit:
IF CamResult3 > 19 THEN
	NokCounter3re := NokCounter3re +1;
END_IF
END_ACTION

ACTION Print_Back_OK__exit:
CamResult3:=CamResult3+10;	(*   0 = noch kein Bild gemacht*)
				(*   1 =  Frontseite OK*)
				(*  11 = Frontseite und Rückseite OK*)
				(*  99 = Teil ist NOK	*)
END_ACTION

ACTION mitte_zu__action:
ST03_422_Y64_6.MoveInit:=TRUE;
END_ACTION

ACTION hinten_auf__action:
ST03_422_Y64_5.MoveInit:=TRUE;
END_ACTION

ACTION ResetNokCounter_entry:
(*Register um eins nach hinten schieben*)
i:=0;
FOR i:=100 TO 2 BY-1 DO
   NokPercent[i] := NokPercent[i-1];
END_FOR

IF	CamResult = 11 AND
	CamResult2 = 11 AND
	CamResult3 = 11 THEN
	NokCounter:=0;
	NokPercent[1] := FALSE;
ELSIF NOT DummyTest_160pol THEN
	gNokPartsColorCam := gNokPartsColorCam+1;
	NokCounter:=NokCounter+1;
	NokPercent[1] := TRUE;
END_IF
END_ACTION

ACTION CheckCounter_entry:
(*Anzahl der Schlechtteile von den letzten 100 Prüfungen*)
i:=0;
NokCounterPercent:=0;
FOR i:=1 TO 100 BY 1 DO
  IF	NokPercent[i] THEN
	NokCounterPercent:=NokCounterPercent+1;
	END_IF
END_FOR
END_ACTION

ACTION Msg_Cam_entry:
MessageHandler.ClearMessageLines(sVisu:=Visu.Message);
END_ACTION

ACTION Msg_Cam_action:
MessageHandler.Msg.ID:='PM112';
MessageHandler.Msg.Name:='Sensopart Kam.-Erg. Prüfung  n.i.o:';
MessageHandler.Msg.Text:='Sensopart Kam.-Erg. Prüfung  n.i.o:';

MessageHandler.Msg.Color:=Color.red;
MessageHandler.Msg.Station:=3;

MessageHandler(
	Prio:=2, 								(*1=highest, .. , 4=lowest*)
	Btn1Addr:=ADR(MsgOk),				(*Address of Button1 , if Zero then Button is unvisible*)
	Btn2Addr:=0(*ADR(MsgCancel)*),			(*Address of Button2 , if Zero then Button is unvisible*)
	sVisu:=Visu.Message);
END_ACTION

ACTION Msg_Cam_exit:
MsgOk:=FALSE;
MsgCancel:=FALSE;
END_ACTION

ACTION Counter_Reset_entry:
NokCounter:=0;
(*Percent Register löschen*)
i:=0;
FOR i:=1 TO 100 BY 1 DO
  NokPercent[i]:= FALSE;
END_FOR
NokCounterPercent:=0;
END_ACTION

ACTION Msg_Cam_Percent_entry:
MessageHandler.ClearMessageLines(sVisu:=Visu.Message);
END_ACTION

ACTION Msg_Cam_Percent_action:
MessageHandler.Msg.ID:='PM113';
MessageHandler.Msg.Name:='Sensopart Kam.-Erg. Prüfung  n.i.o:';
MessageHandler.Msg.Text:='Sensopart Kam.-Erg. Prüfung n.i.o:';

MessageHandler.Msg.Color:=Color.red;
MessageHandler.Msg.Station:=3;

MessageHandler(
	Prio:=2, 								(*1=highest, .. , 4=lowest*)
	Btn1Addr:=ADR(MsgOk),				(*Address of Button1 , if Zero then Button is unvisible*)
	Btn2Addr:=0(*ADR(MsgCancel)*),			(*Address of Button2 , if Zero then Button is unvisible*)
	sVisu:=Visu.Message);
END_ACTION

ACTION Msg_Cam_Percent_exit:
MsgOk:=FALSE;
MsgCancel:=FALSE;
END_ACTION

ACTION Zylinder_3_auf__action:
ST03_423_Y65_7.MoveWork := TRUE;
END_ACTION

ACTION Zylinder_3_auf__exit:
(*Ergebnis Protduktion*)
Result160pol:=CamResult;

IF	CamResult =11 AND
	CamResult2 = 11 AND
	CamResult3 = 11 THEN
	ST03_Main.Result:=RESULT_OK;
ELSE
	ST03_Main.Result:=RESULT_NOK;
END_IF
END_ACTION

ACTION Zylinder_1_zu__action:
ST03_422_Y64_7.MoveWork:=TRUE;
END_ACTION

ACTION SeqEnd_action:
SFCTime:=TIME_TO_DINT(TIME()-SFCTimeStart);
State:=STATE_WAIT;
END_ACTION

TRANSITION OK:
NOT MP.ST03.SGM_3621
OR
ST03_S18.BitInToCheck
END_TRANSITION

TRANSITION OK:
(
ST03_70U3_1.BitInToCheck	 AND	 	(*Bereit/ Im Druck Tintenstrahldrucker Frontseite*)
ST03_71U3_1.BitInToCheck	 AND		 (*Bereit/ Im Druck Tintenstrahldrucker Rückseite*)
NOT ST03_70U3_3.BitInToCheck AND	 (*Fehler/Störung Tintenstrahldrucker Frontseite*)
NOT ST03_71U3_3.BitInToCheck AND	 (*Fehler/Störung Tintenstrahldrucker Rückseite*)
ST03_70U3_2.BitInToCheck AND 		(*Tank voll Tintenstrahldrucker Frontseite*)
ST03_71U3_2.BitInToCheck  			(*Tank voll Tintenstrahldrucker Rückseite*)
) OR
(*b_Printer_Off OR*)
DummyTest_160pol
OR
( MP.ST03.SGM_3621 AND
ST03_70U3_1.BitInToCheck	 AND	 	(*Bereit/ Im Druck Tintenstrahldrucker Frontseite*)
ST03_71U3_1.BitInToCheck	 AND		 (*Bereit/ Im Druck Tintenstrahldrucker Rückseite*)
NOT ST03_70U3_3.BitInToCheck AND	 (*Fehler/Störung Tintenstrahldrucker Frontseite*)
NOT ST03_71U3_3.BitInToCheck )	 (*Fehler/Störung Tintenstrahldrucker Rückseite*)
END_TRANSITION

TRANSITION Front_NOK:
NOT ST03_70U3_1.BitInToCheck	  (*Bereit/ Im Druck Tintenstrahldrucker Frontseite*)
END_TRANSITION

TRANSITION Back_NOK:
NOT ST03_71U3_1.BitInToCheck	  (*Bereit/ Im Druck Tintenstrahldrucker Rückseite*)
END_TRANSITION

TRANSITION TankFront_leer:
NOT MP.ST03.SGM_3621 AND
NOT ST03_70U3_2.BitInToCheck  	(*Tank voll Tintenstrahldrucker Frontseite*)
END_TRANSITION

TRANSITION TankBack_leer:
NOT MP.ST03.SGM_3621 AND
NOT ST03_71U3_2.BitInToCheck  	(*Tank voll Tintenstrahldrucker Rückseite*)
END_TRANSITION

TRANSITION ErrFront:
ST03_70U3_3.BitInToCheck  (*Fehler/Störung Tintenstrahldrucker Frontseite*)
END_TRANSITION

TRANSITION ErrBack:
ST03_71U3_3.BitInToCheck  (*Fehler/Störung Tintenstrahldrucker Rückseite*)
END_TRANSITION

TRANSITION Frontcam_bb:
NOT MP.ST03.FrontCamOn OR
(NOT ST03_8_80_A1.b_kamera_aktiv		 (*Sensopart Kamera Frontseite*)
AND
NOT ST03_8_80_A1.sm_kamera_nicht_bb  (*Sensopart Kamera Frontseite*)
AND
NOT ST03_8_90_A1.sm_kamera_nicht_bb
AND
ST03_8_90_A1.st_ctrl_out.b_bereit
AND
ST03_8_90_A1.Activated)
END_TRANSITION

TRANSITION Backcam_bb:
NOT MP.ST03.BackCamOn OR
(NOT ST03_8_85_A1.b_kamera_aktiv		 (*Sensopart Kamera rechts*)
AND
NOT ST03_8_85_A1.sm_kamera_nicht_bb	 (*Sensopart Kamera rechts*)
AND
NOT ST03_8_95_A1.sm_kamera_nicht_bb	(*Sensopart Kamera Ethernet rechts *)
AND
ST03_8_95_A1.st_ctrl_out.b_bereit			(*Sensopart Kamera Ethernet rechts *)
AND
ST03_8_95_A1.Activated)
END_TRANSITION

TRANSITION Vereinzler_frei:
NOT ST03_421_B63_7.BitInToCheck 			(*  ISK anwesend am Vereinzler*)
END_TRANSITION

TRANSITION StateOk:
ST03_422_Y64_5.State=STATE_OK AND
ST03_422_Y64_6.State=STATE_OK AND
ST03_421_B63_7.BitInToCheck 			(*  ISK anwesend am Vereinzler*)
AND
gTipImp
END_TRANSITION

TRANSITION StateOk:
ST03_422_Y64_5.State=STATE_OK
AND
gTipImp
END_TRANSITION

TRANSITION Print_Cam_free:
NOT ST03_422_B64_3.BitInToCheck	 AND	(* Förderband ISK anwesend Stopper 1 Kamera*)
NOT ST03_423_B65_2.BitInToCheck	AND (* Förderband ISK anwesend Stopper Kamera 2*)
NOT ST03_423_B65_5.BitInToCheck	AND (* Förderband ISK anwesend Stopper 3 Kamera*)
NOT ST03_422_B64_0.BitInToCheck	AND(* Förderband Trigger Tintenstrahldrucker (Lichtschranke 1)*)
NOT ST03_423_B66_0.BitInToCheck	(* Förderband Trigger Tintenstrahldrucker (Lichtschranke 2)*)
AND
gTipImp
END_TRANSITION

TRANSITION StateOk:
ST03_422_Y64_7.State=STATE_OK AND
ST03_422_Y64_6.State=STATE_OK AND
gTipImp
END_TRANSITION

TRANSITION Iso_on_CamPos:
ST03_422_B64_3.BitInToCheck	 (* Förderband ISK anwesend Stopper 1 Kamera*)
AND
gTipImp
END_TRANSITION

TRANSITION aktiv:
ST03_8_80_A1.b_kamera_aktiv OR(*Sensopart Kamera Frontseite*)
ST03_8_90_A1.Activated
END_TRANSITION

TRANSITION Busy:
ST03_8_80_A1.b_busy OR  (*Sensopart Kamera Frontseite*)
ST03_8_90_A1.st_ctrl_out.b_busy
END_TRANSITION

TRANSITION Done:
(ST03_8_80_A1.b_done AND	 (*Sensopart Kamera Frontseite*)(
(ST03_8_80_A1.Ergebnis_IO AND NOT ST03_8_80_A1.Ergebnis_NIO)OR
RepeatCounter>=2 ))
OR
(ST03_8_90_A1.st_ctrl_out.b_fertig AND
((ST03_8_90_A1.b_Kam_Pruef_IO AND NOT ST03_8_90_A1.b_Kam_Pruef_NIO) OR
RepeatCounter>=2))
END_TRANSITION

TRANSITION CamNotAktiv:
(ST03_8_80_A1.b_done	 (*Sensopart Kamera Frontseite*)
AND
NOT MP.ST03.FrontCamOn)
OR
(ST03_8_90_A1.st_ctrl_out.b_fertig  (*Kamera Farberkennung Ethernet*)
AND
NOT MP.ST03.FrontCamOn)
END_TRANSITION

TRANSITION CamDone:
ST03_8_80_A1.b_done	 (*Sensopart Kamera links*)
OR
ST03_8_90_A1.st_ctrl_out.b_fertig	 (*Sensopart Kamera Ethernet links *)
END_TRANSITION

TRANSITION aktiv:
ST03_8_85_A1.b_kamera_aktiv OR 	(*Sensopart Kamera rechts*)
ST03_8_95_A1.Activated			(*Sensopart Kamera Ethernet rechts *)
END_TRANSITION

TRANSITION Busy:
ST03_8_85_A1.b_busy OR				 (*Sensopart Kamera rechts*)
ST03_8_95_A1.st_ctrl_out.b_busy		(*Sensopart Kamera Ethernet rechts *)
END_TRANSITION

TRANSITION Done:
(ST03_8_85_A1.b_done AND		 (*Sensopart Kamera rechts*)
((ST03_8_85_A1.Ergebnis_IO AND NOT ST03_8_85_A1.Ergebnis_NIO)OR
RepeatCounter>=2 ))
OR
(ST03_8_95_A1.st_ctrl_out.b_fertig AND	(*Sensopart Kamera Ethernet rechts *)
((ST03_8_95_A1.b_Kam_Pruef_IO AND NOT ST03_8_95_A1.b_Kam_Pruef_NIO) OR
RepeatCounter>=2))
END_TRANSITION

TRANSITION CamNotAktiv:
(ST03_8_85_A1.b_done				 (*Sensopart Kamera rechts*)
AND
NOT MP.ST03.BackCamOn)
OR
(ST03_8_95_A1.st_ctrl_out.b_fertig 	(*Sensopart Kamera Ethernet rechts *)
AND
NOT MP.ST03.BackCamOn)
END_TRANSITION

TRANSITION CamDone:
ST03_8_85_A1.b_done				 (*Sensopart Kamera rechts*)
OR
ST03_8_95_A1.st_ctrl_out.b_fertig	(*Sensopart Kamera Ethernet rechts *)
END_TRANSITION

TRANSITION StateOk:
ST03_423_Y65_6.State = STATE_OK AND
gTipImp
END_TRANSITION

TRANSITION StateOk:
ST03_422_Y64_7.State = STATE_OK AND
gTipImp
END_TRANSITION

TRANSITION Iso_on_CamPos_2:
ST03_423_B65_2.BitInToCheck	 (* Förderband ISK anwesend Stopper Kamera*)
AND
gTipImp
END_TRANSITION

TRANSITION aktiv:
ST03_8_80_A1.b_kamera_aktiv OR(*Sensopart Kamera Frontseite*)
ST03_8_90_A1.Activated
END_TRANSITION

TRANSITION Busy:
ST03_8_80_A1.b_busy OR  			(*Sensopart Kamera links*)
ST03_8_90_A1.st_ctrl_out.b_busy	 (*Sensopart Kamera Ethernet links *)
END_TRANSITION

TRANSITION Done:
(ST03_8_80_A1.b_done AND		 (*Sensopart Kamera links*)
(
(ST03_8_80_A1.Ergebnis_IO AND NOT ST03_8_80_A1.Ergebnis_NIO)OR
RepeatCounter>=2 ))
OR

(ST03_8_90_A1.st_ctrl_out.b_fertig AND		 (*Sensopart Kamera Ethernet links *)
((ST03_8_90_A1.b_Kam_Pruef_IO AND NOT ST03_8_90_A1.b_Kam_Pruef_NIO) OR
RepeatCounter>=2))
END_TRANSITION

TRANSITION CamNotAktiv:
(ST03_8_80_A1.b_done	 (*Sensopart Kamera links*)
AND
NOT MP.ST03.FrontCamOn)
OR
(ST03_8_90_A1.st_ctrl_out.b_fertig   (*Sensopart Kamera Ethernet links *)
AND
NOT MP.ST03.FrontCamOn)
END_TRANSITION

TRANSITION CamDone:
ST03_8_80_A1.b_done	 (*Sensopart Kamera links*)
OR
ST03_8_90_A1.st_ctrl_out.b_fertig	(*Sensopart Kamera Ethernet links *)
END_TRANSITION

TRANSITION aktiv:
ST03_8_85_A1.b_kamera_aktiv OR 	(*Sensopart Kamera rechts*)
ST03_8_95_A1.Activated			(*Sensopart Kamera Ethernet rechts *)
END_TRANSITION

TRANSITION Busy:
ST03_8_85_A1.b_busy OR			 (*Sensopart Kamera rechts*)
ST03_8_95_A1.st_ctrl_out.b_busy	(*Sensopart Kamera Ethernet rechts *)
END_TRANSITION

TRANSITION Done:
(ST03_8_85_A1.b_done AND				 (*Sensopart Kamera rechts*)
((ST03_8_85_A1.Ergebnis_IO AND NOT ST03_8_85_A1.Ergebnis_NIO)OR
RepeatCounter>=2 ))
OR
(ST03_8_95_A1.st_ctrl_out.b_fertig AND		(*Sensopart Kamera Ethernet rechts *)
((ST03_8_95_A1.b_Kam_Pruef_IO AND NOT ST03_8_95_A1.b_Kam_Pruef_NIO) OR
RepeatCounter>=2))
END_TRANSITION

TRANSITION CamNotAktiv:
(ST03_8_85_A1.b_done	 			(*Sensopart Kamera rechts*)
AND
NOT MP.ST03.BackCamOn)
OR
(ST03_8_95_A1.st_ctrl_out.b_fertig 	(*Sensopart Kamera Ethernet rechts *)
AND
NOT MP.ST03.BackCamOn)
END_TRANSITION

TRANSITION CamDone:
ST03_8_85_A1.b_done				 (*Sensopart Kamera rechts*)
OR
ST03_8_95_A1.st_ctrl_out.b_fertig	 (*Sensopart Kamera Ethernet rechts *)
END_TRANSITION

TRANSITION StateOk:
ST03_423_Y65_7.State = STATE_OK AND
gTipImp
END_TRANSITION

TRANSITION StateOk:
ST03_423_Y65_6.State = STATE_OK AND
gTipImp
END_TRANSITION

TRANSITION Iso_on_CamPos_2:
ST03_423_B65_5.BitInToCheck	 (* Förderband ISK anwesend Stopper Kamera*)
AND
gTipImp
END_TRANSITION

TRANSITION aktiv:
ST03_8_80_A1.b_kamera_aktiv OR	(*Sensopart Kamera links*)
ST03_8_90_A1.Activated			(*Sensopart Kamera Ethernet links *)
END_TRANSITION

TRANSITION Busy:
ST03_8_80_A1.b_busy OR 			 (*Sensopart Kamera links*)
ST03_8_90_A1.st_ctrl_out.b_busy	(*Sensopart Kamera Ethernet links *)
END_TRANSITION

TRANSITION Done:
(ST03_8_80_A1.b_done AND	 (*Sensopart Kamera links*)
(
(ST03_8_80_A1.Ergebnis_IO AND NOT ST03_8_80_A1.Ergebnis_NIO)OR
RepeatCounter>=2 ))
OR
(ST03_8_90_A1.st_ctrl_out.b_fertig AND	(*Sensopart Kamera Ethernet links *)
((ST03_8_90_A1.b_Kam_Pruef_IO AND NOT ST03_8_90_A1.b_Kam_Pruef_NIO) OR
RepeatCounter>=2))
END_TRANSITION

TRANSITION CamNotAktiv:
(ST03_8_80_A1.b_done	 (*Sensopart Kamera links*)
AND
NOT MP.ST03.FrontCamOn)
OR
(ST03_8_90_A1.st_ctrl_out.b_fertig  (*Sensopart Kamera Ethernet links *)
AND
NOT MP.ST03.FrontCamOn)
END_TRANSITION

TRANSITION CamDone:
ST03_8_80_A1.b_done				 (*Sensopart Kamera links*)
OR
ST03_8_90_A1.st_ctrl_out.b_fertig	 (*Sensopart Kamera Ethernet links *)
END_TRANSITION

TRANSITION aktiv:
ST03_8_85_A1.b_kamera_aktiv OR		 (*Sensopart Kamera rechts*)
ST03_8_95_A1.Activated				(*Sensopart Kamera Ethernet rechts *)
END_TRANSITION

TRANSITION Busy:
ST03_8_85_A1.b_busy OR			 (*Sensopart Kamera rechts*)
ST03_8_95_A1.st_ctrl_out.b_busy	(*Sensopart Kamera Ethernet rechts *)
END_TRANSITION

TRANSITION Done:
(ST03_8_85_A1.b_done AND				 (*Sensopart Kamera rechts*)
((ST03_8_85_A1.Ergebnis_IO AND NOT ST03_8_85_A1.Ergebnis_NIO)OR
RepeatCounter>=2 ))
OR
(ST03_8_95_A1.st_ctrl_out.b_fertig AND		(*Sensopart Kamera Ethernet rechts *)
((ST03_8_95_A1.b_Kam_Pruef_IO AND NOT ST03_8_95_A1.b_Kam_Pruef_NIO) OR
RepeatCounter>=2))
END_TRANSITION

TRANSITION CamNotAktiv:
(ST03_8_85_A1.b_done	 			(*Sensopart Kamera rechts*)
AND
NOT MP.ST03.BackCamOn)
OR
(ST03_8_95_A1.st_ctrl_out.b_fertig  (*Sensopart Kamera Ethernet rechts *)
AND
NOT MP.ST03.BackCamOn)
END_TRANSITION

TRANSITION CamDone:
ST03_8_85_A1.b_done	 			(*Sensopart Kamera rechts*)
OR
ST03_8_95_A1.st_ctrl_out.b_fertig	 (*Sensopart Kamera Ethernet rechts *)
END_TRANSITION

TRANSITION StateOk:
ST03_422_Y64_6.State=STATE_OK AND
gTipImp
END_TRANSITION

TRANSITION StateOk:
ST03_422_Y64_5.State=STATE_OK AND
gTipImp
END_TRANSITION

TRANSITION CounterOK:
NokCounter<MP.ST03.CamNoOfErrors AND
NokCounterPercent < MP.ST03.CamNoOfErrorsPercent
END_TRANSITION

TRANSITION Nok_Cont:
NokCounter >= MP.ST03.CamNoOfErrors
END_TRANSITION

TRANSITION Nok_Percent:
NokCounterPercent >= MP.ST03.CamNoOfErrorsPercent
END_TRANSITION

TRANSITION Cam_full:
ST03_423_B65_5.BitInToCheck  (* Förderband ISK anwesend Stopper 3 Kamera*)
END_TRANSITION

TRANSITION free:
NOT ST03_422_B64_4.BitInToCheck AND		(* Zuführung ISK auf Übergabeposition Robo Palettierer*)
ST03_423_B65_5.BitInToCheck		AND			(* Förderband ISK anwesend Stopper Kamera*)
Robot01.ActualArea <> 4
END_TRANSITION

TRANSITION StateOk:
ST03_423_Y65_7.State = STATE_OK AND
ST03_422_B64_4.BitInToCheck AND		(* Zuführung ISK auf Übergabeposition Robo Palettierer*)
NOT ST03_423_B65_5.BitInToCheck		(* Förderband ISK anwesend Stopper Kamera*)
AND
gTipImp
END_TRANSITION

TRANSITION StateOk:
ST03_422_Y64_7.State=STATE_OK
AND
gTipImp
END_TRANSITION
END_PROGRAM

(* POU Stations/ST_03_Ruestsaetze/ST_03_PRGs/ST03_Autostop, ST *)
PROGRAM ST03_Autostop
VAR_INPUT
	Start										:BOOL;
END_VAR
VAR_OUTPUT
END_VAR

VAR
	fb_ton_Autostop						: TON;
	fb_r_trig_Autostop					: R_TRIG;
	Error								: BOOL;
	MsgOK								: BOOL;
END_VAR
fb_ton_Autostop(IN:=Start, PT:=t#500m );
IF	MP.ST00.Override > 0 THEN
	fb_ton_Autostop.PT:=fb_ton_Autostop.PT * (100 / MP.ST00.Override) ;
END_IF

fb_r_trig_Autostop(CLK:=fb_ton_Autostop.Q);
IF	fb_r_trig_Autostop.Q AND
	(gTypeCode=312 OR		 (*nur beim 93 pol*)
	 gTypeCode=4991) THEN 	(*nur beim 102 pol*)
	ModeSelect.iRemoteAutoStop:=TRUE;
	Start:=FALSE;
	Error:=TRUE;
	MessageHandler.ClearMessageLines(sVisu:=Visu.Message);

END_IF

IF	Error THEN
	MessageHandler.Msg.ID:='PM20';
	MessageHandler.Msg.Name:='Timeout';
	MessageHandler.Msg.Text:='Autostop weil die Anlage zu lange gestanden ist!' ;
	MessageHandler.Msg.Color:=Color.yellow;
	MessageHandler.Msg.Station:=0;

	MessageHandler(
		Prio:=2, 							(*1=highest, .. , 4=lowest*)
		Btn1Addr:=ADR(MsgOk),			(*Address of Button1 , if Zero then Button is unvisible*)
		Btn2Addr:=,						(*Address of Button2 , if Zero then Button is unvisible*)
		sVisu:=Visu.Message);

	IF 	MsgOK THEN
		MsgOk:=FALSE;
		Error:=FALSE;
	END_IF

END_IF
END_PROGRAM

